KUKA KRL program: EPS_2_25730_SANINSPMH_A_20250909085212.src

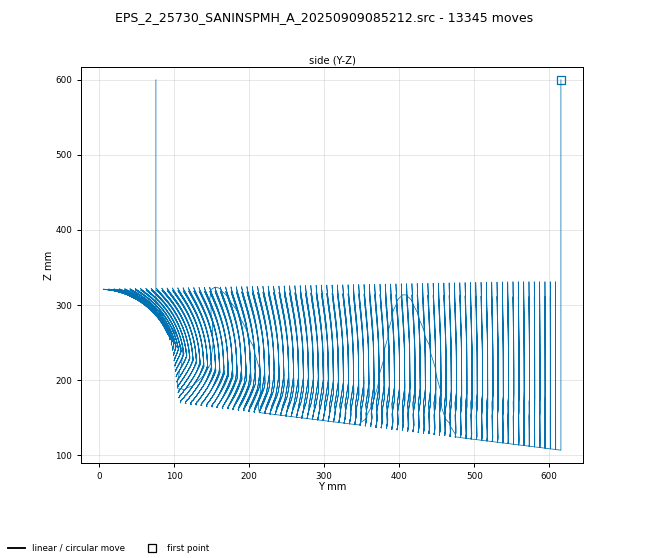
[picture p0: tool path of EPS_2_25730_SANINSPMH_A_20250909085212.src, 13345 of 13347 moves have a stored position in this frame; points joined in program order, loops and branches not executed]
&ACCESS RVP
&REL 4
&COMMENT QRS 19112012
&PARAM EDITMASK = *
DEF PART()
EXT BAS (BAS_COMMAND :IN,REAL :IN )
INT I
BAS (#INITMOV,0 )

;KUKA QRS Post kuka4.cps  Date:22-06-2017 !

File_ID=2820

QRS_PRE_INIT()

;Init var - Until changes are made in qrs_pre_init
Outlet_Square_prg=0
Inlet_1_Square_prg=0
Inlet_2_Square_prg=0
Inlet_3_Square_prg=0
Inlet_4_Square_prg=0
Inlet_5_Square_prg=0

Outlet_1={X 0.000, Y 552.020, Z 256.000, B 0.000, E1 0.000 }
Inlet_1={X 0.000, Y 553.440, Z 236.000, B 0.000, E1 180.000 }
Outlet_1_type=150
Inlet_1_type=150
;QRS#1=Sidecore dimensions
;QRS#2=150-6" PVC SDR 28
;QRS#3=150-6" PVC SDR 28
;QRS#4=
;QRS#5=
;QRS#6=
;QRS#7=
;QRS#8=
;QRS#9=10-06 PSX
;QRS#10=10-06 PSX
;QRS#11=
;QRS#12=
;QRS#13=
;QRS#14=
;QRS#15=
;QRS#16=1220x127x610 2'
;QRS#17=EPS Height
;QRS#18=331
;QRS#19=*
;QRS#20= UPDATED VERSION 22-06-2017
;QRS#21=*
Outlet_Square=070
Inlet_1_Square=070
Inlet_2_Square=0
Inlet_3_Square=0
Inlet_4_Square=0
Inlet_5_Square=0
Mill_Square=1
Outlet_Square_Prg=203
Inlet_1_Square_prg=203

QRS_INIT()

$ADVANCE=5

; T1
PTP {E1 173.612,E2 173.612}
PTP {X 0,Y 615.5,A -85,B 0,C 180,E1 173.612,E2 173.612,E3 0,E4 0,E5 0,E6 0}
QRS_SPEED_INIT()
LIN {X 0,Y 615.5,Z 600,A -85,B 0,C 180,E1 173.612,E2 173.612,E3 0,E4 0,E5 0,E6 0} C_VEL
LIN {X 0,Y 615.5,Z 116.679,A -85,B 0,C 180,E1 173.612,E2 173.612} C_VEL
LIN {X 0,Y 615.5,Z 108.498,A -85,B 0,C 180,E1 173.612,E2 173.612} C_VEL
LIN {X 0,Y 615.484,Z 106.498,A -85,B 0,C 180,E1 173.425,E2 173.425} C_VEL
LIN {X 0,Y 615.477,Z 106.503,A -85,B 0,C 180,E1 170.801,E2 170.801} C_VEL
LIN {X 0,Y 615.484,Z 106.508,A -85,B 0,C 180,E1 168.139,E2 168.139} C_VEL
LIN {X 0,Y 615.491,Z 106.495,A -85,B 0,C 180,E1 165.451,E2 165.451} C_VEL
LIN {X 0,Y 615.489,Z 106.51,A -85,B 0,C 180,E1 162.729,E2 162.729} C_VEL
LIN {X 0,Y 615.481,Z 106.499,A -85,B 0,C 180,E1 159.967,E2 159.967} C_VEL
LIN {X 0,Y 615.481,Z 106.505,A -85,B 0,C 180,E1 157.155,E2 157.155} C_VEL
LIN {X 0,Y 615.477,Z 106.504,A -85,B 0,C 180,E1 154.433,E2 154.433} C_VEL
LIN {X 0,Y 615.485,Z 106.497,A -85,B 0,C 180,E1 152.085,E2 152.085} C_VEL
LIN {X 0,Y 615.489,Z 106.496,A -85,B 0,C 180,E1 149.84,E2 149.84} C_VEL
LIN {X 0,Y 615.481,Z 106.505,A -85,B 0,C 180,E1 147.542,E2 147.542} C_VEL
LIN {X 0,Y 615.495,Z 106.512,A -85,B 0,C 180,E1 145.185,E2 145.185} C_VEL
LIN {X 0,Y 615.472,Z 106.503,A -85,B 0,C 180,E1 142.757,E2 142.757} C_VEL
LIN {X 0,Y 615.483,Z 106.502,A -85,B 0,C 180,E1 139.912,E2 139.912} C_VEL
LIN {X 0,Y 615.491,Z 106.51,A -85,B 0,C 180,E1 137.647,E2 137.647} C_VEL
LIN {X 0,Y 615.474,Z 106.501,A -85,B 0,C 180,E1 134.93,E2 134.93} C_VEL
LIN {X 0,Y 615.482,Z 106.506,A -85,B 0,C 180,E1 132.079,E2 132.079} C_VEL
LIN {X 0,Y 615.491,Z 106.512,A -85,B 0,C 180,E1 129.75,E2 129.75} C_VEL
LIN {X 0,Y 615.48,Z 106.497,A -85,B 0,C 180,E1 126.936,E2 126.936} C_VEL
LIN {X 0,Y 615.492,Z 106.514,A -85,B 0,C 180,E1 124.022,E2 124.022} C_VEL
LIN {X 0,Y 615.472,Z 106.506,A -85,B 0,C 180,E1 121.686,E2 121.686} C_VEL
LIN {X 0,Y 615.473,Z 106.5,A -85,B 0,C 180,E1 119.407,E2 119.407} C_VEL
LIN {X 0,Y 615.493,Z 106.51,A -85,B 0,C 180,E1 116.444,E2 116.444} C_VEL
LIN {X 0,Y 615.472,Z 106.506,A -85,B 0,C 180,E1 114.005,E2 114.005} C_VEL
LIN {X 0,Y 615.485,Z 106.496,A -85,B 0,C 180,E1 111.432,E2 111.432} C_VEL
LIN {X 0,Y 615.499,Z 106.666,A -85,B 0,C 180,E1 108.545,E2 108.545} C_VEL
LIN {X 0,Y 615.476,Z 120.496,A -85,B 0,C 180,E1 105.906,E2 105.906} C_VEL
LIN {X 0,Y 615.489,Z 134.92,A -85,B 0,C 180,E1 103.201,E2 103.201} C_VEL
LIN {X 0,Y 615.474,Z 149.332,A -85,B 0,C 180,E1 100.527,E2 100.527} C_VEL
LIN {X 0,Y 615.496,Z 152.049,A -85,B 0,C 180,E1 100.091,E2 100.091} C_VEL
LIN {X 0,Y 615.495,Z 154.32,A -85,B 0,C 180,E1 100.028,E2 100.028} C_VEL
LIN {X 0,Y 615.496,Z 227.7,A -85,B 0,C 180,E1 99.157,E2 99.157} C_VEL
LIN {X 0,Y 615.497,Z 235.887,A -85,B 0,C 180,E1 98.992,E2 98.992} C_VEL
LIN {X 0,Y 615.497,Z 244.447,A -85,B 0,C 180,E1 98.743,E2 98.743} C_VEL
LIN {X 0,Y 615.497,Z 252.059,A -85,B 0,C 180,E1 98.454,E2 98.454} C_VEL
LIN {X 0,Y 615.499,Z 260.579,A -85,B 0,C 180,E1 98.041,E2 98.041} C_VEL
LIN {X 0,Y 615.489,Z 268.747,A -85,B 0,C 180,E1 97.546,E2 97.546} C_VEL
LIN {X 0,Y 615.492,Z 275.387,A -85,B 0,C 180,E1 97.058,E2 97.058} C_VEL
LIN {X 0,Y 615.498,Z 281.183,A -85,B 0,C 180,E1 96.557,E2 96.557} C_VEL
LIN {X 0,Y 615.499,Z 287.533,A -85,B 0,C 180,E1 95.899,E2 95.899} C_VEL
LIN {X 0,Y 615.495,Z 293.983,A -85,B 0,C 180,E1 95.077,E2 95.077} C_VEL
LIN {X 0,Y 615.491,Z 299.122,A -85,B 0,C 180,E1 94.257,E2 94.257} C_VEL
LIN {X 0,Y 615.493,Z 303.886,A -85,B 0,C 180,E1 93.273,E2 93.273} C_VEL
LIN {X 0,Y 615.493,Z 306.2,A -85,B 0,C 180,E1 92.618,E2 92.618} C_VEL
LIN {X 0,Y 615.499,Z 307.976,A -85,B 0,C 180,E1 91.963,E2 91.963} C_VEL
LIN {X 0,Y 615.492,Z 309.266,A -85,B 0,C 180,E1 91.309,E2 91.309} C_VEL
LIN {X 0,Y 615.491,Z 310.083,A -85,B 0,C 180,E1 90.654,E2 90.654} C_VEL
LIN {X 0,Y 615.492,Z 310.384,A -85,B 0,C 180,E1 90,E2 90} C_VEL
LIN {X 0,Y 615.492,Z 310.125,A -85,B 0,C 180,E1 89.346,E2 89.346} C_VEL
LIN {X 0,Y 615.494,Z 309.394,A -85,B 0,C 180,E1 88.692,E2 88.692} C_VEL
LIN {X 0,Y 615.499,Z 308.195,A -85,B 0,C 180,E1 88.037,E2 88.037} C_VEL
LIN {X 0,Y 615.49,Z 305.377,A -85,B 0,C 180,E1 87.055,E2 87.055} C_VEL
LIN {X 0,Y 615.492,Z 302.81,A -85,B 0,C 180,E1 86.4,E2 86.4} C_VEL
LIN {X 0,Y 615.495,Z 297.744,A -85,B 0,C 180,E1 85.416,E2 85.416} C_VEL
LIN {X 0,Y 615.496,Z 292.289,A -85,B 0,C 180,E1 84.595,E2 84.595} C_VEL
LIN {X 0,Y 615.497,Z 285.454,A -85,B 0,C 180,E1 83.773,E2 83.773} C_VEL
LIN {X 0,Y 615.497,Z 278.42,A -85,B 0,C 180,E1 83.1,E2 83.1} C_VEL
LIN {X 0,Y 615.491,Z 270.073,A -85,B 0,C 180,E1 82.455,E2 82.455} C_VEL
LIN {X 0,Y 615.499,Z 262.197,A -85,B 0,C 180,E1 81.96,E2 81.96} C_VEL
LIN {X 0,Y 615.497,Z 254.076,A -85,B 0,C 180,E1 81.546,E2 81.546} C_VEL
LIN {X 0,Y 615.497,Z 245.865,A -85,B 0,C 180,E1 81.216,E2 81.216} C_VEL
LIN {X 0,Y 615.497,Z 237.842,A -85,B 0,C 180,E1 80.967,E2 80.967} C_VEL
LIN {X 0,Y 615.5,Z 228.165,A -85,B 0,C 180,E1 80.76,E2 80.76} C_VEL
LIN {X 0,Y 615.494,Z 152.561,A -85,B 0,C 180,E1 79.847,E2 79.847} C_VEL
LIN {X 0,Y 615.489,Z 151.218,A -85,B 0,C 180,E1 79.723,E2 79.723} C_VEL
LIN {X 0,Y 615.475,Z 137.207,A -85,B 0,C 180,E1 77.134,E2 77.134} C_VEL
LIN {X 0,Y 615.486,Z 122.781,A -85,B 0,C 180,E1 74.435,E2 74.435} C_VEL
LIN {X 0,Y 615.497,Z 108.44,A -85,B 0,C 180,E1 71.719,E2 71.719} C_VEL
LIN {X 0,Y 615.493,Z 106.562,A -85,B 0,C 180,E1 71.311,E2 71.311} C_VEL
LIN {X 0,Y 615.484,Z 106.497,A -85,B 0,C 180,E1 68.568,E2 68.568} C_VEL
LIN {X 0,Y 615.48,Z 106.51,A -85,B 0,C 180,E1 65.728,E2 65.728} C_VEL
LIN {X 0,Y 615.486,Z 106.497,A -85,B 0,C 180,E1 62.823,E2 62.823} C_VEL
LIN {X 0,Y 615.467,Z 106.506,A -85,B 0,C 180,E1 60.209,E2 60.209} C_VEL
LIN {X 0,Y 615.488,Z 106.506,A -85,B 0,C 180,E1 57.543,E2 57.543} C_VEL
LIN {X 0,Y 615.496,Z 106.495,A -85,B 0,C 180,E1 55.186,E2 55.186} C_VEL
LIN {X 0,Y 615.468,Z 106.501,A -85,B 0,C 180,E1 52.757,E2 52.757} C_VEL
LIN {X 0,Y 615.49,Z 106.508,A -85,B 0,C 180,E1 49.911,E2 49.911} C_VEL
LIN {X 0,Y 615.469,Z 106.502,A -85,B 0,C 180,E1 46.955,E2 46.955} C_VEL
LIN {X 0,Y 615.49,Z 106.508,A -85,B 0,C 180,E1 44.149,E2 44.149} C_VEL
LIN {X 0,Y 615.485,Z 106.496,A -85,B 0,C 180,E1 41.474,E2 41.474} C_VEL
LIN {X 0,Y 615.475,Z 106.507,A -85,B 0,C 180,E1 38.905,E2 38.905} C_VEL
LIN {X 0,Y 615.484,Z 106.509,A -85,B 0,C 180,E1 36.425,E2 36.425} C_VEL
LIN {X 0,Y 615.487,Z 106.498,A -85,B 0,C 180,E1 34.022,E2 34.022} C_VEL
LIN {X 0,Y 615.481,Z 106.498,A -85,B 0,C 180,E1 31.686,E2 31.686} C_VEL
LIN {X 0,Y 615.473,Z 106.504,A -85,B 0,C 180,E1 29.407,E2 29.407} C_VEL
LIN {X 0,Y 615.493,Z 106.512,A -85,B 0,C 180,E1 27.047,E2 27.047} C_VEL
LIN {X 0,Y 615.485,Z 106.496,A -85,B 0,C 180,E1 24.008,E2 24.008} C_VEL
LIN {X 0,Y 615.483,Z 106.509,A -85,B 0,C 180,E1 21.432,E2 21.432} C_VEL
LIN {X 0,Y 615.486,Z 106.498,A -85,B 0,C 180,E1 18.605,E2 18.605} C_VEL
LIN {X 0,Y 615.474,Z 106.504,A -85,B 0,C 180,E1 15.906,E2 15.906} C_VEL
LIN {X 0,Y 615.479,Z 106.507,A -85,B 0,C 180,E1 13.201,E2 13.201} C_VEL
LIN {X 0,Y 615.486,Z 106.496,A -85,B 0,C 180,E1 10.527,E2 10.527} C_VEL
LIN {X 0,Y 615.486,Z 106.51,A -85,B 0,C 180,E1 7.876,E2 7.876} C_VEL
LIN {X 0,Y 615.479,Z 106.501,A -85,B 0,C 180,E1 5.241,E2 5.241} C_VEL
LIN {X 0,Y 615.482,Z 106.499,A -85,B 0,C 180,E1 2.618,E2 2.618} C_VEL
LIN {X 0,Y 615.487,Z 106.515,A -85,B 0,C 180,E1 0,E2 0} C_VEL
LIN {X 0,Y 615.481,Z 106.499,A -85,B 0,C 180,E1 -2.618,E2 -2.618} C_VEL
LIN {X 0,Y 615.481,Z 106.502,A -85,B 0,C 180,E1 -5.241,E2 -5.241} C_VEL
LIN {X 0,Y 615.485,Z 106.509,A -85,B 0,C 180,E1 -7.876,E2 -7.876} C_VEL
LIN {X 0,Y 615.485,Z 106.496,A -85,B 0,C 180,E1 -10.527,E2 -10.527} C_VEL
LIN {X 0,Y 615.485,Z 106.507,A -85,B 0,C 180,E1 -13.201,E2 -13.201} C_VEL
LIN {X 0,Y 615.474,Z 106.503,A -85,B 0,C 180,E1 -15.905,E2 -15.905} C_VEL
LIN {X 0,Y 615.486,Z 106.499,A -85,B 0,C 180,E1 -18.646,E2 -18.646} C_VEL
LIN {X 0,Y 615.479,Z 106.508,A -85,B 0,C 180,E1 -21.432,E2 -21.432} C_VEL
LIN {X 0,Y 615.489,Z 106.496,A -85,B 0,C 180,E1 -24.272,E2 -24.272} C_VEL
LIN {X 0,Y 615.477,Z 106.51,A -85,B 0,C 180,E1 -27.178,E2 -27.178} C_VEL
LIN {X 0,Y 615.482,Z 106.497,A -85,B 0,C 180,E1 -29.794,E2 -29.794} C_VEL
LIN {X 0,Y 615.486,Z 106.506,A -85,B 0,C 180,E1 -32.457,E2 -32.457} C_VEL
LIN {X 0,Y 615.485,Z 106.51,A -85,B 0,C 180,E1 -34.815,E2 -34.815} C_VEL
LIN {X 0,Y 615.469,Z 106.502,A -85,B 0,C 180,E1 -37.243,E2 -37.243} C_VEL
LIN {X 0,Y 615.486,Z 106.504,A -85,B 0,C 180,E1 -40.089,E2 -40.089} C_VEL
LIN {X 0,Y 615.499,Z 106.513,A -85,B 0,C 180,E1 -42.352,E2 -42.352} C_VEL
LIN {X 0,Y 615.47,Z 106.5,A -85,B 0,C 180,E1 -45.07,E2 -45.07} C_VEL
LIN {X 0,Y 615.49,Z 106.507,A -85,B 0,C 180,E1 -47.919,E2 -47.919} C_VEL
LIN {X 0,Y 615.48,Z 106.51,A -85,B 0,C 180,E1 -50.25,E2 -50.25} C_VEL
LIN {X 0,Y 615.478,Z 106.498,A -85,B 0,C 180,E1 -53.064,E2 -53.064} C_VEL
LIN {X 0,Y 615.485,Z 106.511,A -85,B 0,C 180,E1 -55.978,E2 -55.978} C_VEL
LIN {X 0,Y 615.461,Z 106.506,A -85,B 0,C 180,E1 -58.313,E2 -58.313} C_VEL
LIN {X 0,Y 615.469,Z 106.5,A -85,B 0,C 180,E1 -60.593,E2 -60.593} C_VEL
LIN {X 0,Y 615.497,Z 106.497,A -85,B 0,C 180,E1 -62.953,E2 -62.953} C_VEL
LIN {X 0,Y 615.475,Z 106.509,A -85,B 0,C 180,E1 -65.728,E2 -65.728} C_VEL
LIN {X 0,Y 615.463,Z 106.507,A -85,B 0,C 180,E1 -67.863,E2 -67.863} C_VEL
LIN {X 0,Y 615.494,Z 106.696,A -85,B 0,C 180,E1 -69.398,E2 -69.398} C_VEL
LIN {X 0,Y 615.489,Z 122.513,A -85,B 0,C 180,E1 -72.043,E2 -72.043} C_VEL
LIN {X 0,Y 615.468,Z 140.241,A -85,B 0,C 180,E1 -74.943,E2 -74.943} C_VEL
LIN {X 0,Y 615.465,Z 155.869,A -85,B 0,C 180,E1 -77.47,E2 -77.47} C_VEL
LIN {X 0,Y 615.491,Z 170.941,A -85,B 0,C 180,E1 -79.847,E2 -79.847} C_VEL
LIN {X 0,Y 615.489,Z 172.866,A -85,B 0,C 180,E1 -79.91,E2 -79.91} C_VEL
LIN {X 0,Y 615.493,Z 247.945,A -85,B 0,C 180,E1 -80.801,E2 -80.801} C_VEL
LIN {X 0,Y 615.496,Z 257.699,A -85,B 0,C 180,E1 -81.009,E2 -81.009} C_VEL
LIN {X 0,Y 615.499,Z 268.156,A -85,B 0,C 180,E1 -81.34,E2 -81.34} C_VEL
LIN {X 0,Y 615.497,Z 278.43,A -85,B 0,C 180,E1 -81.794,E2 -81.794} C_VEL
LIN {X 0,Y 615.493,Z 288.2,A -85,B 0,C 180,E1 -82.372,E2 -82.372} C_VEL
LIN {X 0,Y 615.494,Z 295.936,A -85,B 0,C 180,E1 -82.942,E2 -82.942} C_VEL
LIN {X 0,Y 615.497,Z 303.336,A -85,B 0,C 180,E1 -83.608,E2 -83.608} C_VEL
LIN {X 0,Y 615.498,Z 310.739,A -85,B 0,C 180,E1 -84.43,E2 -84.43} C_VEL
LIN {X 0,Y 615.497,Z 316.534,A -85,B 0,C 180,E1 -85.252,E2 -85.252} C_VEL
LIN {X 0,Y 615.496,Z 321.101,A -85,B 0,C 180,E1 -86.072,E2 -86.072} C_VEL
LIN {X 0,Y 615.492,Z 324.069,A -85,B 0,C 180,E1 -86.727,E2 -86.727} C_VEL
LIN {X 0,Y 615.494,Z 326.357,A -85,B 0,C 180,E1 -87.382,E2 -87.382} C_VEL
LIN {X 0,Y 615.499,Z 328.085,A -85,B 0,C 180,E1 -88.037,E2 -88.037} C_VEL
LIN {X 0,Y 615.493,Z 329.33,A -85,B 0,C 180,E1 -88.692,E2 -88.692} C_VEL
LIN {X 0,Y 615.491,Z 330.104,A -85,B 0,C 180,E1 -89.346,E2 -89.346} C_VEL
LIN {X 0,Y 615.491,Z 330.389,A -85,B 0,C 180,E1 -90,E2 -90} C_VEL
LIN {X 0,Y 615.492,Z 330.104,A -85,B 0,C 180,E1 -90.654,E2 -90.654} C_VEL
LIN {X 0,Y 615.493,Z 329.33,A -85,B 0,C 180,E1 -91.309,E2 -91.309} C_VEL
LIN {X 0,Y 615.499,Z 328.085,A -85,B 0,C 180,E1 -91.963,E2 -91.963} C_VEL
LIN {X 0,Y 615.488,Z 325.22,A -85,B 0,C 180,E1 -92.946,E2 -92.946} C_VEL
LIN {X 0,Y 615.491,Z 322.603,A -85,B 0,C 180,E1 -93.601,E2 -93.601} C_VEL
LIN {X 0,Y 615.495,Z 317.481,A -85,B 0,C 180,E1 -94.585,E2 -94.585} C_VEL
LIN {X 0,Y 615.495,Z 311.967,A -85,B 0,C 180,E1 -95.406,E2 -95.406} C_VEL
LIN {X 0,Y 615.498,Z 305.016,A -85,B 0,C 180,E1 -96.228,E2 -96.228} C_VEL
LIN {X 0,Y 615.496,Z 297.858,A -85,B 0,C 180,E1 -96.901,E2 -96.901} C_VEL
LIN {X 0,Y 615.488,Z 290.619,A -85,B 0,C 180,E1 -97.463,E2 -97.463} C_VEL
LIN {X 0,Y 615.498,Z 282.865,A -85,B 0,C 180,E1 -97.958,E2 -97.958} C_VEL
LIN {X 0,Y 615.498,Z 274.91,A -85,B 0,C 180,E1 -98.371,E2 -98.371} C_VEL
LIN {X 0,Y 615.497,Z 265.75,A -85,B 0,C 180,E1 -98.743,E2 -98.743} C_VEL
LIN {X 0,Y 615.496,Z 257.686,A -85,B 0,C 180,E1 -98.992,E2 -98.992} C_VEL
LIN {X 0,Y 615.493,Z 247.925,A -85,B 0,C 180,E1 -99.199,E2 -99.199} C_VEL
LIN {X 0,Y 615.49,Z 171.745,A -85,B 0,C 180,E1 -100.111,E2 -100.111} C_VEL
LIN {X 0,Y 615.489,Z 170.51,A -85,B 0,C 180,E1 -100.194,E2 -100.194} C_VEL
LIN {X 0,Y 615.49,Z 153.783,A -85,B 0,C 180,E1 -102.866,E2 -102.866} C_VEL
LIN {X 0,Y 615.481,Z 136.068,A -85,B 0,C 180,E1 -105.735,E2 -105.735} C_VEL
LIN {X 0,Y 615.487,Z 120.566,A -85,B 0,C 180,E1 -108.278,E2 -108.278} C_VEL
LIN {X 0,Y 615.494,Z 106.695,A -85,B 0,C 180,E1 -110.602,E2 -110.602} C_VEL
LIN {X 0,Y 615.491,Z 106.506,A -85,B 0,C 180,E1 -112.844,E2 -112.844} C_VEL
LIN {X 0,Y 615.461,Z 106.503,A -85,B 0,C 180,E1 -115.717,E2 -115.717} C_VEL
LIN {X 0,Y 615.497,Z 106.511,A -85,B 0,C 180,E1 -118.452,E2 -118.452} C_VEL
LIN {X 0,Y 615.48,Z 106.498,A -85,B 0,C 180,E1 -121.085,E2 -121.085} C_VEL
LIN {X 0,Y 615.463,Z 106.504,A -85,B 0,C 180,E1 -123.531,E2 -123.531} C_VEL
LIN {X 0,Y 615.475,Z 106.509,A -85,B 0,C 180,E1 -125.832,E2 -125.832} C_VEL
LIN {X 0,Y 615.488,Z 106.514,A -85,B 0,C 180,E1 -128.069,E2 -128.069} C_VEL
LIN {X 0,Y 615.487,Z 106.498,A -85,B 0,C 180,E1 -130.607,E2 -130.607} C_VEL
LIN {X 0,Y 615.465,Z 106.504,A -85,B 0,C 180,E1 -133.247,E2 -133.247} C_VEL
LIN {X 0,Y 615.489,Z 106.506,A -85,B 0,C 180,E1 -136.003,E2 -136.003} C_VEL
LIN {X 0,Y 615.484,Z 106.497,A -85,B 0,C 180,E1 -138.526,E2 -138.526} C_VEL
LIN {X 0,Y 615.47,Z 106.506,A -85,B 0,C 180,E1 -141.094,E2 -141.094} C_VEL
LIN {X 0,Y 615.486,Z 106.511,A -85,B 0,C 180,E1 -143.575,E2 -143.575} C_VEL
LIN {X 0,Y 615.474,Z 106.499,A -85,B 0,C 180,E1 -146.468,E2 -146.468} C_VEL
LIN {X 0,Y 615.486,Z 106.51,A -85,B 0,C 180,E1 -149.08,E2 -149.08} C_VEL
LIN {X 0,Y 615.483,Z 106.497,A -85,B 0,C 180,E1 -152.085,E2 -152.085} C_VEL
LIN {X 0,Y 615.492,Z 106.514,A -85,B 0,C 180,E1 -155.009,E2 -155.009} C_VEL
LIN {X 0,Y 615.485,Z 106.496,A -85,B 0,C 180,E1 -157.864,E2 -157.864} C_VEL
LIN {X 0,Y 615.488,Z 106.51,A -85,B 0,C 180,E1 -160.662,E2 -160.662} C_VEL
LIN {X 0,Y 615.488,Z 106.496,A -85,B 0,C 180,E1 -163.569,E2 -163.569} C_VEL
LIN {X 0,Y 615.473,Z 106.505,A -85,B 0,C 180,E1 -166.126,E2 -166.126} C_VEL
LIN {X 0,Y 615.485,Z 106.506,A -85,B 0,C 180,E1 -168.807,E2 -168.807} C_VEL
LIN {X 0,Y 615.486,Z 106.496,A -85,B 0,C 180,E1 -171.463,E2 -171.463} C_VEL
LIN {X 0,Y 615.485,Z 106.509,A -85,B 0,C 180,E1 -174.102,E2 -174.102} C_VEL
LIN {X 0,Y 615.479,Z 106.502,A -85,B 0,C 180,E1 -176.727,E2 -176.727} C_VEL
LIN {X 0,Y 615.479,Z 106.499,A -85,B 0,C 180,E1 -179.346,E2 -179.346} C_VEL
LIN {X 0,Y 615.496,Z 106.512,A -85,B 0,C 180,E1 -181.963,E2 -181.963} C_VEL
LIN {X 0,Y 615.484,Z 106.498,A -85,B 0,C 180,E1 -184.585,E2 -184.585} C_VEL
LIN {X 0,Y 615.484,Z 106.498,A -85,B 0,C 180,E1 -186.575,E2 -186.575} C_VEL
LIN {X 0,Y 614.803,Z 106.649,A -85,B 0,C 180,E1 -187.121,E2 -187.121} C_VEL
LIN {X 0,Y 611.964,Z 107.069,A -85,B 0,C 180,E1 -188.007,E2 -188.007} C_VEL
LIN {X 0,Y 609.574,Z 107.378,A -85,B 0,C 180,E1 -188.719,E2 -188.719} C_VEL
LIN {X 0,Y 608.543,Z 107.494,A -85,B 0,C 180,E1 -189.269,E2 -189.269} C_VEL
LIN {X 0,Y 608.455,Z 107.503,A -85,B 0,C 180,E1 -189.455,E2 -189.455} C_VEL
LIN {X 0,Y 608.462,Z 107.503,A -85,B 0,C 180,E1 -192,E2 -192} C_VEL
LIN {X 0,Y 608.478,Z 107.498,A -85,B 0,C 180,E1 -194.721,E2 -194.721} C_VEL
LIN {X 0,Y 608.453,Z 107.51,A -85,B 0,C 180,E1 -197.477,E2 -197.477} C_VEL
LIN {X 0,Y 608.46,Z 107.499,A -85,B 0,C 180,E1 -200.274,E2 -200.274} C_VEL
LIN {X 0,Y 608.46,Z 107.5,A -85,B 0,C 180,E1 -202.476,E2 -202.476} C_VEL
LIN {X 0,Y 608.456,Z 107.502,A -85,B 0,C 180,E1 -204.571,E2 -204.571} C_VEL
LIN {X 0,Y 608.484,Z 107.504,A -85,B 0,C 180,E1 -207.208,E2 -207.208} C_VEL
LIN {X 0,Y 608.467,Z 107.498,A -85,B 0,C 180,E1 -209.971,E2 -209.971} C_VEL
LIN {X 0,Y 608.452,Z 107.51,A -85,B 0,C 180,E1 -212.88,E2 -212.88} C_VEL
LIN {X 0,Y 608.444,Z 107.504,A -85,B 0,C 180,E1 -215.278,E2 -215.278} C_VEL
LIN {X 0,Y 608.464,Z 107.503,A -85,B 0,C 180,E1 -218.24,E2 -218.24} C_VEL
LIN {X 0,Y 608.456,Z 107.5,A -85,B 0,C 180,E1 -221.342,E2 -221.342} C_VEL
LIN {X 0,Y 608.452,Z 107.508,A -85,B 0,C 180,E1 -224.263,E2 -224.263} C_VEL
LIN {X 0,Y 608.441,Z 107.502,A -85,B 0,C 180,E1 -227.039,E2 -227.039} C_VEL
LIN {X 0,Y 608.454,Z 107.503,A -85,B 0,C 180,E1 -229.697,E2 -229.697} C_VEL
LIN {X 0,Y 608.465,Z 107.506,A -85,B 0,C 180,E1 -232.253,E2 -232.253} C_VEL
LIN {X 0,Y 608.485,Z 107.496,A -85,B 0,C 180,E1 -235.09,E2 -235.09} C_VEL
LIN {X 0,Y 608.464,Z 107.509,A -85,B 0,C 180,E1 -237.905,E2 -237.905} C_VEL
LIN {X 0,Y 608.458,Z 107.503,A -85,B 0,C 180,E1 -240.22,E2 -240.22} C_VEL
LIN {X 0,Y 608.482,Z 107.497,A -85,B 0,C 180,E1 -242.792,E2 -242.792} C_VEL
LIN {X 0,Y 608.472,Z 107.504,A -85,B 0,C 180,E1 -245.849,E2 -245.849} C_VEL
LIN {X 0,Y 608.464,Z 107.499,A -85,B 0,C 180,E1 -248.308,E2 -248.308} C_VEL
LIN {X 0,Y 608.49,Z 107.574,A -85,B 0,C 180,E1 -251.379,E2 -251.379} C_VEL
LIN {X 0,Y 608.48,Z 120.639,A -85,B 0,C 180,E1 -253.907,E2 -253.907} C_VEL
LIN {X 0,Y 608.477,Z 135.127,A -85,B 0,C 180,E1 -256.644,E2 -256.644} C_VEL
LIN {X 0,Y 608.424,Z 149.617,A -85,B 0,C 180,E1 -259.349,E2 -259.349} C_VEL
LIN {X 0,Y 608.471,Z 152.233,A -85,B 0,C 180,E1 -259.792,E2 -259.792} C_VEL
LIN {X 0,Y 608.525,Z 154.822,A -85,B 0,C 180,E1 -259.856,E2 -259.856} C_VEL
LIN {X 0,Y 608.511,Z 228.245,A -85,B 0,C 180,E1 -260.737,E2 -260.737} C_VEL
LIN {X 0,Y 608.512,Z 237.948,A -85,B 0,C 180,E1 -260.946,E2 -260.946} C_VEL
LIN {X 0,Y 608.499,Z 249.535,A -85,B 0,C 180,E1 -261.323,E2 -261.323} C_VEL
LIN {X 0,Y 608.479,Z 259.431,A -85,B 0,C 180,E1 -261.782,E2 -261.782} C_VEL
LIN {X 0,Y 608.473,Z 267.884,A -85,B 0,C 180,E1 -262.283,E2 -262.283} C_VEL
LIN {X 0,Y 608.46,Z 275.853,A -85,B 0,C 180,E1 -262.867,E2 -262.867} C_VEL
LIN {X 0,Y 608.467,Z 282.902,A -85,B 0,C 180,E1 -263.496,E2 -263.496} C_VEL
LIN {X 0,Y 608.458,Z 289.394,A -85,B 0,C 180,E1 -264.199,E2 -264.199} C_VEL
LIN {X 0,Y 608.437,Z 295.641,A -85,B 0,C 180,E1 -265.03,E2 -265.03} C_VEL
LIN {X 0,Y 608.434,Z 301.424,A -85,B 0,C 180,E1 -266.026,E2 -266.026} C_VEL
LIN {X 0,Y 608.447,Z 305.63,A -85,B 0,C 180,E1 -267.02,E2 -267.02} C_VEL
LIN {X 0,Y 608.443,Z 308.569,A -85,B 0,C 180,E1 -268.014,E2 -268.014} C_VEL
LIN {X 0,Y 608.445,Z 309.87,A -85,B 0,C 180,E1 -268.676,E2 -268.676} C_VEL
LIN {X 0,Y 608.434,Z 310.692,A -85,B 0,C 180,E1 -269.338,E2 -269.338} C_VEL
LIN {X 0,Y 608.432,Z 310.995,A -85,B 0,C 180,E1 -270,E2 -270} C_VEL
LIN {X 0,Y 608.435,Z 310.735,A -85,B 0,C 180,E1 -270.662,E2 -270.662} C_VEL
LIN {X 0,Y 608.446,Z 309.998,A -85,B 0,C 180,E1 -271.324,E2 -271.324} C_VEL
LIN {X 0,Y 608.443,Z 308.787,A -85,B 0,C 180,E1 -271.986,E2 -271.986} C_VEL
LIN {X 0,Y 608.445,Z 305.942,A -85,B 0,C 180,E1 -272.979,E2 -272.979} C_VEL
LIN {X 0,Y 608.446,Z 303.353,A -85,B 0,C 180,E1 -273.642,E2 -273.642} C_VEL
LIN {X 0,Y 608.445,Z 298.245,A -85,B 0,C 180,E1 -274.638,E2 -274.638} C_VEL
LIN {X 0,Y 608.461,Z 292.75,A -85,B 0,C 180,E1 -275.468,E2 -275.468} C_VEL
LIN {X 0,Y 608.454,Z 285.15,A -85,B 0,C 180,E1 -276.374,E2 -276.374} C_VEL
LIN {X 0,Y 608.463,Z 276.951,A -85,B 0,C 180,E1 -277.132,E2 -277.132} C_VEL
LIN {X 0,Y 608.473,Z 269.202,A -85,B 0,C 180,E1 -277.716,E2 -277.716} C_VEL
LIN {X 0,Y 608.48,Z 261.037,A -85,B 0,C 180,E1 -278.217,E2 -278.217} C_VEL
LIN {X 0,Y 608.484,Z 250.677,A -85,B 0,C 180,E1 -278.719,E2 -278.719} C_VEL
LIN {X 0,Y 608.511,Z 239.038,A -85,B 0,C 180,E1 -279.116,E2 -279.116} C_VEL
LIN {X 0,Y 608.524,Z 228.648,A -85,B 0,C 180,E1 -279.347,E2 -279.347} C_VEL
LIN {X 0,Y 608.514,Z 189.347,A -85,B 0,C 180,E1 -279.829,E2 -279.829} C_VEL
LIN {X 0,Y 608.489,Z 152.717,A -85,B 0,C 180,E1 -280.271,E2 -280.271} C_VEL
LIN {X 0,Y 608.456,Z 151.482,A -85,B 0,C 180,E1 -280.397,E2 -280.397} C_VEL
LIN {X 0,Y 608.447,Z 137.42,A -85,B 0,C 180,E1 -283.017,E2 -283.017} C_VEL
LIN {X 0,Y 608.456,Z 122.926,A -85,B 0,C 180,E1 -285.75,E2 -285.75} C_VEL
LIN {X 0,Y 608.491,Z 107.915,A -85,B 0,C 180,E1 -288.622,E2 -288.622} C_VEL
LIN {X 0,Y 608.462,Z 107.507,A -85,B 0,C 180,E1 -288.869,E2 -288.869} C_VEL
LIN {X 0,Y 608.461,Z 107.499,A -85,B 0,C 180,E1 -291.692,E2 -291.692} C_VEL
LIN {X 0,Y 608.453,Z 107.509,A -85,B 0,C 180,E1 -294.571,E2 -294.571} C_VEL
LIN {X 0,Y 608.443,Z 107.502,A -85,B 0,C 180,E1 -297.518,E2 -297.518} C_VEL
LIN {X 0,Y 608.457,Z 107.505,A -85,B 0,C 180,E1 -299.97,E2 -299.97} C_VEL
LIN {X 0,Y 608.452,Z 107.501,A -85,B 0,C 180,E1 -302.88,E2 -302.88} C_VEL
LIN {X 0,Y 608.437,Z 107.503,A -85,B 0,C 180,E1 -305.278,E2 -305.278} C_VEL
LIN {X 0,Y 608.467,Z 107.504,A -85,B 0,C 180,E1 -308.24,E2 -308.24} C_VEL
LIN {X 0,Y 608.449,Z 107.503,A -85,B 0,C 180,E1 -311.341,E2 -311.341} C_VEL
LIN {X 0,Y 608.453,Z 107.503,A -85,B 0,C 180,E1 -314.263,E2 -314.263} C_VEL
LIN {X 0,Y 608.44,Z 107.504,A -85,B 0,C 180,E1 -317.039,E2 -317.039} C_VEL
LIN {X 0,Y 608.451,Z 107.508,A -85,B 0,C 180,E1 -319.696,E2 -319.696} C_VEL
LIN {X 0,Y 608.465,Z 107.499,A -85,B 0,C 180,E1 -322.253,E2 -322.253} C_VEL
LIN {X 0,Y 608.443,Z 107.503,A -85,B 0,C 180,E1 -324.722,E2 -324.722} C_VEL
LIN {X 0,Y 608.459,Z 107.505,A -85,B 0,C 180,E1 -327.478,E2 -327.478} C_VEL
LIN {X 0,Y 608.468,Z 107.498,A -85,B 0,C 180,E1 -330.22,E2 -330.22} C_VEL
LIN {X 0,Y 608.479,Z 107.503,A -85,B 0,C 180,E1 -332.792,E2 -332.792} C_VEL
LIN {X 0,Y 608.479,Z 107.497,A -85,B 0,C 180,E1 -335.847,E2 -335.847} C_VEL
LIN {X 0,Y 608.467,Z 107.501,A -85,B 0,C 180,E1 -338.308,E2 -338.308} C_VEL
LIN {X 0,Y 608.47,Z 107.5,A -85,B 0,C 180,E1 -341.283,E2 -341.283} C_VEL
LIN {X 0,Y 608.454,Z 107.501,A -85,B 0,C 180,E1 -343.906,E2 -343.906} C_VEL
LIN {X 0,Y 608.457,Z 107.507,A -85,B 0,C 180,E1 -346.643,E2 -346.643} C_VEL
LIN {X 0,Y 608.464,Z 107.499,A -85,B 0,C 180,E1 -349.35,E2 -349.35} C_VEL
LIN {X 0,Y 608.477,Z 107.503,A -85,B 0,C 180,E1 -352.033,E2 -352.033} C_VEL
LIN {X 0,Y 608.46,Z 107.502,A -85,B 0,C 180,E1 -354.698,E2 -354.698} C_VEL
LIN {X 0,Y 608.473,Z 107.499,A -85,B 0,C 180,E1 -357.352,E2 -357.352} C_VEL
LIN {X 0,Y 608.477,Z 107.507,A -85,B 0,C 180,E1 -360,E2 -360} C_VEL
LIN {X 0,Y 608.472,Z 107.498,A -85,B 0,C 180,E1 -362.648,E2 -362.648} C_VEL
LIN {X 0,Y 608.461,Z 107.502,A -85,B 0,C 180,E1 -365.302,E2 -365.302} C_VEL
LIN {X 0,Y 608.477,Z 107.503,A -85,B 0,C 180,E1 -367.967,E2 -367.967} C_VEL
LIN {X 0,Y 608.468,Z 107.5,A -85,B 0,C 180,E1 -370.956,E2 -370.956} C_VEL
LIN {X 0,Y 608.46,Z 107.508,A -85,B 0,C 180,E1 -373.356,E2 -373.356} C_VEL
LIN {X 0,Y 608.454,Z 107.501,A -85,B 0,C 180,E1 -376.094,E2 -376.094} C_VEL
LIN {X 0,Y 608.456,Z 107.504,A -85,B 0,C 180,E1 -378.87,E2 -378.87} C_VEL
LIN {X 0,Y 608.464,Z 107.501,A -85,B 0,C 180,E1 -381.692,E2 -381.692} C_VEL
LIN {X 0,Y 608.457,Z 107.503,A -85,B 0,C 180,E1 -384.571,E2 -384.571} C_VEL
LIN {X 0,Y 608.444,Z 107.503,A -85,B 0,C 180,E1 -387.518,E2 -387.518} C_VEL
LIN {X 0,Y 608.466,Z 107.499,A -85,B 0,C 180,E1 -389.972,E2 -389.972} C_VEL
LIN {X 0,Y 608.45,Z 107.508,A -85,B 0,C 180,E1 -392.88,E2 -392.88} C_VEL
LIN {X 0,Y 608.439,Z 107.503,A -85,B 0,C 180,E1 -395.278,E2 -395.278} C_VEL
LIN {X 0,Y 608.466,Z 107.504,A -85,B 0,C 180,E1 -398.241,E2 -398.241} C_VEL
LIN {X 0,Y 608.454,Z 107.5,A -85,B 0,C 180,E1 -401.342,E2 -401.342} C_VEL
LIN {X 0,Y 608.459,Z 107.51,A -85,B 0,C 180,E1 -404.264,E2 -404.264} C_VEL
LIN {X 0,Y 608.437,Z 107.502,A -85,B 0,C 180,E1 -407.039,E2 -407.039} C_VEL
LIN {X 0,Y 608.456,Z 107.504,A -85,B 0,C 180,E1 -409.697,E2 -409.697} C_VEL
LIN {X 0,Y 608.462,Z 107.505,A -85,B 0,C 180,E1 -412.254,E2 -412.254} C_VEL
LIN {X 0,Y 608.484,Z 107.497,A -85,B 0,C 180,E1 -415.09,E2 -415.09} C_VEL
LIN {X 0,Y 608.464,Z 107.507,A -85,B 0,C 180,E1 -417.906,E2 -417.906} C_VEL
LIN {X 0,Y 608.449,Z 107.503,A -85,B 0,C 180,E1 -420.22,E2 -420.22} C_VEL
LIN {X 0,Y 608.481,Z 107.497,A -85,B 0,C 180,E1 -422.792,E2 -422.792} C_VEL
LIN {X 0,Y 608.462,Z 107.502,A -85,B 0,C 180,E1 -425.851,E2 -425.851} C_VEL
LIN {X 0,Y 608.459,Z 107.501,A -85,B 0,C 180,E1 -428.308,E2 -428.308} C_VEL
LIN {X 0,Y 608.506,Z 107.66,A -85,B 0,C 180,E1 -429.312,E2 -429.312} C_VEL
LIN {X 0,Y 608.486,Z 122.58,A -85,B 0,C 180,E1 -431.83,E2 -431.83} C_VEL
LIN {X 0,Y 608.482,Z 139.321,A -85,B 0,C 180,E1 -434.595,E2 -434.595} C_VEL
LIN {X 0,Y 608.446,Z 156.062,A -85,B 0,C 180,E1 -437.323,E2 -437.323} C_VEL
LIN {X 0,Y 608.467,Z 171.122,A -85,B 0,C 180,E1 -439.729,E2 -439.729} C_VEL
LIN {X 0,Y 608.517,Z 173.315,A -85,B 0,C 180,E1 -439.793,E2 -439.793} C_VEL
LIN {X 0,Y 608.504,Z 247.155,A -85,B 0,C 180,E1 -440.674,E2 -440.674} C_VEL
LIN {X 0,Y 608.522,Z 256.421,A -85,B 0,C 180,E1 -440.863,E2 -440.863} C_VEL
LIN {X 0,Y 608.489,Z 264.893,A -85,B 0,C 180,E1 -441.114,E2 -441.114} C_VEL
LIN {X 0,Y 608.502,Z 273.393,A -85,B 0,C 180,E1 -441.448,E2 -441.448} C_VEL
LIN {X 0,Y 608.497,Z 281.723,A -85,B 0,C 180,E1 -441.866,E2 -441.866} C_VEL
LIN {X 0,Y 608.472,Z 289.762,A -85,B 0,C 180,E1 -442.367,E2 -442.367} C_VEL
LIN {X 0,Y 608.453,Z 297.417,A -85,B 0,C 180,E1 -442.951,E2 -442.951} C_VEL
LIN {X 0,Y 608.452,Z 305.439,A -85,B 0,C 180,E1 -443.7,E2 -443.7} C_VEL
LIN {X 0,Y 608.46,Z 312.431,A -85,B 0,C 180,E1 -444.532,E2 -444.532} C_VEL
LIN {X 0,Y 608.431,Z 317.986,A -85,B 0,C 180,E1 -445.362,E2 -445.362} C_VEL
LIN {X 0,Y 608.445,Z 323.147,A -85,B 0,C 180,E1 -446.358,E2 -446.358} C_VEL
LIN {X 0,Y 608.444,Z 325.786,A -85,B 0,C 180,E1 -447.021,E2 -447.021} C_VEL
LIN {X 0,Y 608.443,Z 328.679,A -85,B 0,C 180,E1 -448.014,E2 -448.014} C_VEL
LIN {X 0,Y 608.445,Z 329.934,A -85,B 0,C 180,E1 -448.676,E2 -448.676} C_VEL
LIN {X 0,Y 608.434,Z 330.714,A -85,B 0,C 180,E1 -449.338,E2 -449.338} C_VEL
LIN {X 0,Y 608.431,Z 331,A -85,B 0,C 180,E1 -450,E2 -450} C_VEL
LIN {X 0,Y 608.434,Z 330.714,A -85,B 0,C 180,E1 -450.662,E2 -450.662} C_VEL
LIN {X 0,Y 608.445,Z 329.933,A -85,B 0,C 180,E1 -451.324,E2 -451.324} C_VEL
LIN {X 0,Y 608.443,Z 328.678,A -85,B 0,C 180,E1 -451.986,E2 -451.986} C_VEL
LIN {X 0,Y 608.444,Z 325.785,A -85,B 0,C 180,E1 -452.98,E2 -452.98} C_VEL
LIN {X 0,Y 608.445,Z 323.145,A -85,B 0,C 180,E1 -453.643,E2 -453.643} C_VEL
LIN {X 0,Y 608.431,Z 317.984,A -85,B 0,C 180,E1 -454.638,E2 -454.638} C_VEL
LIN {X 0,Y 608.46,Z 312.429,A -85,B 0,C 180,E1 -455.468,E2 -455.468} C_VEL
LIN {X 0,Y 608.455,Z 304.67,A -85,B 0,C 180,E1 -456.376,E2 -456.376} C_VEL
LIN {X 0,Y 608.453,Z 297.413,A -85,B 0,C 180,E1 -457.05,E2 -457.05} C_VEL
LIN {X 0,Y 608.472,Z 289.758,A -85,B 0,C 180,E1 -457.633,E2 -457.633} C_VEL
LIN {X 0,Y 608.497,Z 281.717,A -85,B 0,C 180,E1 -458.134,E2 -458.134} C_VEL
LIN {X 0,Y 608.502,Z 273.386,A -85,B 0,C 180,E1 -458.552,E2 -458.552} C_VEL
LIN {X 0,Y 608.49,Z 264.884,A -85,B 0,C 180,E1 -458.887,E2 -458.887} C_VEL
LIN {X 0,Y 608.512,Z 255.578,A -85,B 0,C 180,E1 -459.159,E2 -459.159} C_VEL
LIN {X 0,Y 608.51,Z 244.538,A -85,B 0,C 180,E1 -459.368,E2 -459.368} C_VEL
LIN {X 0,Y 608.508,Z 171.945,A -85,B 0,C 180,E1 -460.229,E2 -460.229} C_VEL
LIN {X 0,Y 608.452,Z 170.757,A -85,B 0,C 180,E1 -460.314,E2 -460.314} C_VEL
LIN {X 0,Y 608.483,Z 152.921,A -85,B 0,C 180,E1 -463.186,E2 -463.186} C_VEL
LIN {X 0,Y 608.464,Z 135.134,A -85,B 0,C 180,E1 -466.094,E2 -466.094} C_VEL
LIN {X 0,Y 608.481,Z 119.291,A -85,B 0,C 180,E1 -468.719,E2 -468.719} C_VEL
LIN {X 0,Y 608.488,Z 107.561,A -85,B 0,C 180,E1 -470.725,E2 -470.725} C_VEL
LIN {X 0,Y 608.448,Z 107.502,A -85,B 0,C 180,E1 -473.124,E2 -473.124} C_VEL
LIN {X 0,Y 608.453,Z 107.501,A -85,B 0,C 180,E1 -475.717,E2 -475.717} C_VEL
LIN {X 0,Y 608.45,Z 107.509,A -85,B 0,C 180,E1 -478.267,E2 -478.267} C_VEL
LIN {X 0,Y 608.472,Z 107.504,A -85,B 0,C 180,E1 -480.545,E2 -480.545} C_VEL
LIN {X 0,Y 608.452,Z 107.502,A -85,B 0,C 180,E1 -482.88,E2 -482.88} C_VEL
LIN {X 0,Y 608.435,Z 107.503,A -85,B 0,C 180,E1 -485.278,E2 -485.278} C_VEL
LIN {X 0,Y 608.468,Z 107.505,A -85,B 0,C 180,E1 -488.24,E2 -488.24} C_VEL
LIN {X 0,Y 608.436,Z 107.503,A -85,B 0,C 180,E1 -491.178,E2 -491.178} C_VEL
LIN {X 0,Y 608.47,Z 107.507,A -85,B 0,C 180,E1 -493.869,E2 -493.869} C_VEL
LIN {X 0,Y 608.464,Z 107.499,A -85,B 0,C 180,E1 -496.692,E2 -496.692} C_VEL
LIN {X 0,Y 608.44,Z 107.502,A -85,B 0,C 180,E1 -498.822,E2 -498.822} C_VEL
LIN {X 0,Y 608.466,Z 107.505,A -85,B 0,C 180,E1 -501.76,E2 -501.76} C_VEL
LIN {X 0,Y 608.439,Z 107.503,A -85,B 0,C 180,E1 -504.722,E2 -504.722} C_VEL
LIN {X 0,Y 608.462,Z 107.506,A -85,B 0,C 180,E1 -507.478,E2 -507.478} C_VEL
LIN {X 0,Y 608.467,Z 107.498,A -85,B 0,C 180,E1 -510.22,E2 -510.22} C_VEL
LIN {X 0,Y 608.475,Z 107.503,A -85,B 0,C 180,E1 -512.794,E2 -512.794} C_VEL
LIN {X 0,Y 608.479,Z 107.497,A -85,B 0,C 180,E1 -515.847,E2 -515.847} C_VEL
LIN {X 0,Y 608.463,Z 107.501,A -85,B 0,C 180,E1 -518.308,E2 -518.308} C_VEL
LIN {X 0,Y 608.472,Z 107.5,A -85,B 0,C 180,E1 -521.284,E2 -521.284} C_VEL
LIN {X 0,Y 608.453,Z 107.501,A -85,B 0,C 180,E1 -523.906,E2 -523.906} C_VEL
LIN {X 0,Y 608.462,Z 107.508,A -85,B 0,C 180,E1 -526.644,E2 -526.644} C_VEL
LIN {X 0,Y 608.464,Z 107.499,A -85,B 0,C 180,E1 -529.35,E2 -529.35} C_VEL
LIN {X 0,Y 608.475,Z 107.502,A -85,B 0,C 180,E1 -532.033,E2 -532.033} C_VEL
LIN {X 0,Y 608.462,Z 107.503,A -85,B 0,C 180,E1 -534.698,E2 -534.698} C_VEL
LIN {X 0,Y 608.472,Z 107.498,A -85,B 0,C 180,E1 -537.352,E2 -537.352} C_VEL
LIN {X 0,Y 608.477,Z 107.506,A -85,B 0,C 180,E1 -540,E2 -540} C_VEL
LIN {X 0,Y 608.473,Z 107.499,A -85,B 0,C 180,E1 -542.648,E2 -542.648} C_VEL
LIN {X 0,Y 608.457,Z 107.502,A -85,B 0,C 180,E1 -545.302,E2 -545.302} C_VEL
LIN {X 0,Y 608.479,Z 107.504,A -85,B 0,C 180,E1 -547.967,E2 -547.967} C_VEL
LIN {X 0,Y 608.455,Z 107.503,A -85,B 0,C 180,E1 -549.455,E2 -549.455} C_VEL
LIN {X 0,Y 607.781,Z 107.59,A -85,B 0,C 180,E1 -550.008,E2 -550.008} C_VEL
LIN {X 0,Y 604.929,Z 107.943,A -85,B 0,C 180,E1 -550.905,E2 -550.905} C_VEL
LIN {X 0,Y 602.525,Z 108.249,A -85,B 0,C 180,E1 -551.626,E2 -551.626} C_VEL
LIN {X 0,Y 601.494,Z 108.37,A -85,B 0,C 180,E1 -552.183,E2 -552.183} C_VEL
LIN {X 0,Y 601.41,Z 108.378,A -85,B 0,C 180,E1 -552.371,E2 -552.371} C_VEL
LIN {X 0,Y 601.431,Z 108.377,A -85,B 0,C 180,E1 -554.897,E2 -554.897} C_VEL
LIN {X 0,Y 601.433,Z 108.378,A -85,B 0,C 180,E1 -556.986,E2 -556.986} C_VEL
LIN {X 0,Y 601.405,Z 108.381,A -85,B 0,C 180,E1 -559.81,E2 -559.81} C_VEL
LIN {X 0,Y 601.413,Z 108.379,A -85,B 0,C 180,E1 -562.683,E2 -562.683} C_VEL
LIN {X 0,Y 601.403,Z 108.384,A -85,B 0,C 180,E1 -564.879,E2 -564.879} C_VEL
LIN {X 0,Y 601.42,Z 108.381,A -85,B 0,C 180,E1 -567.363,E2 -567.363} C_VEL
LIN {X 0,Y 601.43,Z 108.376,A -85,B 0,C 180,E1 -570.164,E2 -570.164} C_VEL
LIN {X 0,Y 601.418,Z 108.385,A -85,B 0,C 180,E1 -572.715,E2 -572.715} C_VEL
LIN {X 0,Y 601.403,Z 108.383,A -85,B 0,C 180,E1 -575.113,E2 -575.113} C_VEL
LIN {X 0,Y 601.434,Z 108.375,A -85,B 0,C 180,E1 -577.419,E2 -577.419} C_VEL
LIN {X 0,Y 601.404,Z 108.38,A -85,B 0,C 180,E1 -579.996,E2 -579.996} C_VEL
LIN {X 0,Y 601.41,Z 108.384,A -85,B 0,C 180,E1 -582.671,E2 -582.671} C_VEL
LIN {X 0,Y 601.4,Z 108.379,A -85,B 0,C 180,E1 -585.479,E2 -585.479} C_VEL
LIN {X 0,Y 601.42,Z 108.384,A -85,B 0,C 180,E1 -588.407,E2 -588.407} C_VEL
LIN {X 0,Y 601.41,Z 108.378,A -85,B 0,C 180,E1 -590.873,E2 -590.873} C_VEL
LIN {X 0,Y 601.406,Z 108.379,A -85,B 0,C 180,E1 -593.417,E2 -593.417} C_VEL
LIN {X 0,Y 601.419,Z 108.385,A -85,B 0,C 180,E1 -596.066,E2 -596.066} C_VEL
LIN {X 0,Y 601.419,Z 108.378,A -85,B 0,C 180,E1 -598.546,E2 -598.546} C_VEL
LIN {X 0,Y 601.432,Z 108.379,A -85,B 0,C 180,E1 -601.373,E2 -601.373} C_VEL
LIN {X 0,Y 601.404,Z 108.388,A -85,B 0,C 180,E1 -603.636,E2 -603.636} C_VEL
LIN {X 0,Y 601.45,Z 108.378,A -85,B 0,C 180,E1 -605.859,E2 -605.859} C_VEL
LIN {X 0,Y 601.406,Z 108.379,A -85,B 0,C 180,E1 -608.761,E2 -608.761} C_VEL
LIN {X 0,Y 601.484,Z 108.566,A -85,B 0,C 180,E1 -611.364,E2 -611.364} C_VEL
LIN {X 0,Y 601.421,Z 122.453,A -85,B 0,C 180,E1 -614.061,E2 -614.061} C_VEL
LIN {X 0,Y 601.402,Z 136.941,A -85,B 0,C 180,E1 -616.828,E2 -616.828} C_VEL
LIN {X 0,Y 601.405,Z 151.999,A -85,B 0,C 180,E1 -619.649,E2 -619.649} C_VEL
LIN {X 0,Y 601.518,Z 153.318,A -85,B 0,C 180,E1 -619.715,E2 -619.715} C_VEL
LIN {X 0,Y 601.506,Z 228.279,A -85,B 0,C 180,E1 -620.628,E2 -620.628} C_VEL
LIN {X 0,Y 601.488,Z 238.803,A -85,B 0,C 180,E1 -620.861,E2 -620.861} C_VEL
LIN {X 0,Y 601.473,Z 250.536,A -85,B 0,C 180,E1 -621.263,E2 -621.263} C_VEL
LIN {X 0,Y 601.455,Z 260.931,A -85,B 0,C 180,E1 -621.77,E2 -621.77} C_VEL
LIN {X 0,Y 601.437,Z 269.114,A -85,B 0,C 180,E1 -622.277,E2 -622.277} C_VEL
LIN {X 0,Y 601.414,Z 276.875,A -85,B 0,C 180,E1 -622.868,E2 -622.868} C_VEL
LIN {X 0,Y 601.394,Z 284.708,A -85,B 0,C 180,E1 -623.598,E2 -623.598} C_VEL
LIN {X 0,Y 601.383,Z 292.114,A -85,B 0,C 180,E1 -624.467,E2 -624.467} C_VEL
LIN {X 0,Y 601.34,Z 297.728,A -85,B 0,C 180,E1 -625.307,E2 -625.307} C_VEL
LIN {X 0,Y 601.366,Z 302.943,A -85,B 0,C 180,E1 -626.315,E2 -626.315} C_VEL
LIN {X 0,Y 601.345,Z 305.633,A -85,B 0,C 180,E1 -626.985,E2 -626.985} C_VEL
LIN {X 0,Y 601.342,Z 308.572,A -85,B 0,C 180,E1 -627.991,E2 -627.991} C_VEL
LIN {X 0,Y 601.345,Z 309.871,A -85,B 0,C 180,E1 -628.66,E2 -628.66} C_VEL
LIN {X 0,Y 601.335,Z 310.692,A -85,B 0,C 180,E1 -629.33,E2 -629.33} C_VEL
LIN {X 0,Y 601.333,Z 310.996,A -85,B 0,C 180,E1 -630,E2 -630} C_VEL
LIN {X 0,Y 601.336,Z 310.735,A -85,B 0,C 180,E1 -630.669,E2 -630.669} C_VEL
LIN {X 0,Y 601.346,Z 309.998,A -85,B 0,C 180,E1 -631.339,E2 -631.339} C_VEL
LIN {X 0,Y 601.342,Z 308.788,A -85,B 0,C 180,E1 -632.009,E2 -632.009} C_VEL
LIN {X 0,Y 601.344,Z 305.942,A -85,B 0,C 180,E1 -633.015,E2 -633.015} C_VEL
LIN {X 0,Y 601.365,Z 303.351,A -85,B 0,C 180,E1 -633.685,E2 -633.685} C_VEL
LIN {X 0,Y 601.362,Z 298.243,A -85,B 0,C 180,E1 -634.692,E2 -634.692} C_VEL
LIN {X 0,Y 601.384,Z 292.747,A -85,B 0,C 180,E1 -635.532,E2 -635.532} C_VEL
LIN {X 0,Y 601.394,Z 284.589,A -85,B 0,C 180,E1 -636.504,E2 -636.504} C_VEL
LIN {X 0,Y 601.414,Z 276.947,A -85,B 0,C 180,E1 -637.217,E2 -637.217} C_VEL
LIN {X 0,Y 601.416,Z 269.198,A -85,B 0,C 180,E1 -637.807,E2 -637.807} C_VEL
LIN {X 0,Y 601.447,Z 261.033,A -85,B 0,C 180,E1 -638.314,E2 -638.314} C_VEL
LIN {X 0,Y 601.461,Z 250.662,A -85,B 0,C 180,E1 -638.822,E2 -638.822} C_VEL
LIN {X 0,Y 601.493,Z 239.021,A -85,B 0,C 180,E1 -639.224,E2 -639.224} C_VEL
LIN {X 0,Y 601.518,Z 228.616,A -85,B 0,C 180,E1 -639.457,E2 -639.457} C_VEL
LIN {X 0,Y 601.553,Z 180.357,A -85,B 0,C 180,E1 -640.05,E2 -640.05} C_VEL
LIN {X 0,Y 601.44,Z 152.687,A -85,B 0,C 180,E1 -640.392,E2 -640.392} C_VEL
LIN {X 0,Y 601.384,Z 151.478,A -85,B 0,C 180,E1 -640.521,E2 -640.521} C_VEL
LIN {X 0,Y 601.4,Z 137.417,A -85,B 0,C 180,E1 -643.172,E2 -643.172} C_VEL
LIN {X 0,Y 601.418,Z 124.734,A -85,B 0,C 180,E1 -645.591,E2 -645.591} C_VEL
LIN {X 0,Y 601.484,Z 110.239,A -85,B 0,C 180,E1 -648.39,E2 -648.39} C_VEL
LIN {X 0,Y 601.428,Z 108.436,A -85,B 0,C 180,E1 -648.778,E2 -648.778} C_VEL
LIN {X 0,Y 601.406,Z 108.38,A -85,B 0,C 180,E1 -651.239,E2 -651.239} C_VEL
LIN {X 0,Y 601.444,Z 108.378,A -85,B 0,C 180,E1 -654.141,E2 -654.141} C_VEL
LIN {X 0,Y 601.455,Z 108.373,A -85,B 0,C 180,E1 -657.111,E2 -657.111} C_VEL
LIN {X 0,Y 601.41,Z 108.378,A -85,B 0,C 180,E1 -659.393,E2 -659.393} C_VEL
LIN {X 0,Y 601.4,Z 108.382,A -85,B 0,C 180,E1 -661.727,E2 -661.727} C_VEL
LIN {X 0,Y 601.422,Z 108.387,A -85,B 0,C 180,E1 -664.118,E2 -664.118} C_VEL
LIN {X 0,Y 601.405,Z 108.38,A -85,B 0,C 180,E1 -666.583,E2 -666.583} C_VEL
LIN {X 0,Y 601.408,Z 108.378,A -85,B 0,C 180,E1 -669.126,E2 -669.126} C_VEL
LIN {X 0,Y 601.422,Z 108.386,A -85,B 0,C 180,E1 -671.765,E2 -671.765} C_VEL
LIN {X 0,Y 601.396,Z 108.38,A -85,B 0,C 180,E1 -674.532,E2 -674.532} C_VEL
LIN {X 0,Y 601.413,Z 108.384,A -85,B 0,C 180,E1 -677.409,E2 -677.409} C_VEL
LIN {X 0,Y 601.402,Z 108.381,A -85,B 0,C 180,E1 -680.004,E2 -680.004} C_VEL
LIN {X 0,Y 601.432,Z 108.375,A -85,B 0,C 180,E1 -682.618,E2 -682.618} C_VEL
LIN {X 0,Y 601.414,Z 108.383,A -85,B 0,C 180,E1 -685.068,E2 -685.068} C_VEL
LIN {X 0,Y 601.428,Z 108.381,A -85,B 0,C 180,E1 -687.484,E2 -687.484} C_VEL
LIN {X 0,Y 601.428,Z 108.376,A -85,B 0,C 180,E1 -689.851,E2 -689.851} C_VEL
LIN {X 0,Y 601.417,Z 108.381,A -85,B 0,C 180,E1 -692.637,E2 -692.637} C_VEL
LIN {X 0,Y 601.403,Z 108.385,A -85,B 0,C 180,E1 -695.121,E2 -695.121} C_VEL
LIN {X 0,Y 601.414,Z 108.379,A -85,B 0,C 180,E1 -697.394,E2 -697.394} C_VEL
LIN {X 0,Y 601.405,Z 108.38,A -85,B 0,C 180,E1 -700.19,E2 -700.19} C_VEL
LIN {X 0,Y 601.433,Z 108.379,A -85,B 0,C 180,E1 -703.014,E2 -703.014} C_VEL
LIN {X 0,Y 601.42,Z 108.378,A -85,B 0,C 180,E1 -705.908,E2 -705.908} C_VEL
LIN {X 0,Y 601.432,Z 108.383,A -85,B 0,C 180,E1 -708.542,E2 -708.542} C_VEL
LIN {X 0,Y 601.415,Z 108.377,A -85,B 0,C 180,E1 -711.262,E2 -711.262} C_VEL
LIN {X 0,Y 601.417,Z 108.383,A -85,B 0,C 180,E1 -713.963,E2 -713.963} C_VEL
LIN {X 0,Y 601.422,Z 108.378,A -85,B 0,C 180,E1 -716.65,E2 -716.65} C_VEL
LIN {X 0,Y 601.448,Z 108.374,A -85,B 0,C 180,E1 -719.33,E2 -719.33} C_VEL
LIN {X 0,Y 601.433,Z 108.383,A -85,B 0,C 180,E1 -722.009,E2 -722.009} C_VEL
LIN {X 0,Y 601.42,Z 108.377,A -85,B 0,C 180,E1 -724.692,E2 -724.692} C_VEL
LIN {X 0,Y 601.438,Z 108.379,A -85,B 0,C 180,E1 -727.385,E2 -727.385} C_VEL
LIN {X 0,Y 601.431,Z 108.378,A -85,B 0,C 180,E1 -730.095,E2 -730.095} C_VEL
LIN {X 0,Y 601.422,Z 108.377,A -85,B 0,C 180,E1 -732.828,E2 -732.828} C_VEL
LIN {X 0,Y 601.411,Z 108.384,A -85,B 0,C 180,E1 -735.591,E2 -735.591} C_VEL
LIN {X 0,Y 601.416,Z 108.377,A -85,B 0,C 180,E1 -738.392,E2 -738.392} C_VEL
LIN {X 0,Y 601.404,Z 108.387,A -85,B 0,C 180,E1 -741.239,E2 -741.239} C_VEL
LIN {X 0,Y 601.457,Z 108.372,A -85,B 0,C 180,E1 -744.14,E2 -744.14} C_VEL
LIN {X 0,Y 601.447,Z 108.38,A -85,B 0,C 180,E1 -747.111,E2 -747.111} C_VEL
LIN {X 0,Y 601.416,Z 108.379,A -85,B 0,C 180,E1 -749.393,E2 -749.393} C_VEL
LIN {X 0,Y 601.399,Z 108.379,A -85,B 0,C 180,E1 -751.727,E2 -751.727} C_VEL
LIN {X 0,Y 601.429,Z 108.377,A -85,B 0,C 180,E1 -754.118,E2 -754.118} C_VEL
LIN {X 0,Y 601.406,Z 108.388,A -85,B 0,C 180,E1 -756.583,E2 -756.583} C_VEL
LIN {X 0,Y 601.408,Z 108.379,A -85,B 0,C 180,E1 -759.127,E2 -759.127} C_VEL
LIN {X 0,Y 601.423,Z 108.378,A -85,B 0,C 180,E1 -761.765,E2 -761.765} C_VEL
LIN {X 0,Y 601.423,Z 108.382,A -85,B 0,C 180,E1 -764.535,E2 -764.535} C_VEL
LIN {X 0,Y 601.41,Z 108.378,A -85,B 0,C 180,E1 -767.409,E2 -767.409} C_VEL
LIN {X 0,Y 601.402,Z 108.388,A -85,B 0,C 180,E1 -770.005,E2 -770.005} C_VEL
LIN {X 0,Y 601.431,Z 108.376,A -85,B 0,C 180,E1 -772.618,E2 -772.618} C_VEL
LIN {X 0,Y 601.439,Z 108.374,A -85,B 0,C 180,E1 -775.07,E2 -775.07} C_VEL
LIN {X 0,Y 601.434,Z 108.38,A -85,B 0,C 180,E1 -777.485,E2 -777.485} C_VEL
LIN {X 0,Y 601.426,Z 108.383,A -85,B 0,C 180,E1 -779.852,E2 -779.852} C_VEL
LIN {X 0,Y 601.414,Z 108.377,A -85,B 0,C 180,E1 -782.638,E2 -782.638} C_VEL
LIN {X 0,Y 601.398,Z 108.383,A -85,B 0,C 180,E1 -785.121,E2 -785.121} C_VEL
LIN {X 0,Y 601.403,Z 108.382,A -85,B 0,C 180,E1 -788.041,E2 -788.041} C_VEL
LIN {X 0,Y 601.451,Z 108.499,A -85,B 0,C 180,E1 -789.197,E2 -789.197} C_VEL
LIN {X 0,Y 601.504,Z 119.889,A -85,B 0,C 180,E1 -791.157,E2 -791.157} C_VEL
LIN {X 0,Y 601.443,Z 136.182,A -85,B 0,C 180,E1 -793.888,E2 -793.888} C_VEL
LIN {X 0,Y 601.44,Z 152.923,A -85,B 0,C 180,E1 -796.657,E2 -796.657} C_VEL
LIN {X 0,Y 601.378,Z 169.664,A -85,B 0,C 180,E1 -799.394,E2 -799.394} C_VEL
LIN {X 0,Y 601.425,Z 171.415,A -85,B 0,C 180,E1 -799.629,E2 -799.629} C_VEL
LIN {X 0,Y 601.531,Z 180.469,A -85,B 0,C 180,E1 -799.758,E2 -799.758} C_VEL
LIN {X 0,Y 601.524,Z 248.453,A -85,B 0,C 180,E1 -800.586,E2 -800.586} C_VEL
LIN {X 0,Y 601.51,Z 258.912,A -85,B 0,C 180,E1 -800.819,E2 -800.819} C_VEL
LIN {X 0,Y 601.472,Z 269.62,A -85,B 0,C 180,E1 -801.178,E2 -801.178} C_VEL
LIN {X 0,Y 601.446,Z 280.24,A -85,B 0,C 180,E1 -801.686,E2 -801.686} C_VEL
LIN {X 0,Y 601.416,Z 288.547,A -85,B 0,C 180,E1 -802.193,E2 -802.193} C_VEL
LIN {X 0,Y 601.412,Z 296.404,A -85,B 0,C 180,E1 -802.783,E2 -802.783} C_VEL
LIN {X 0,Y 601.411,Z 303.598,A -85,B 0,C 180,E1 -803.443,E2 -803.443} C_VEL
LIN {X 0,Y 601.391,Z 311.192,A -85,B 0,C 180,E1 -804.299,E2 -804.299} C_VEL
LIN {X 0,Y 601.38,Z 317.029,A -85,B 0,C 180,E1 -805.14,E2 -805.14} C_VEL
LIN {X 0,Y 601.345,Z 321.632,A -85,B 0,C 180,E1 -805.979,E2 -805.979} C_VEL
LIN {X 0,Y 601.343,Z 324.622,A -85,B 0,C 180,E1 -806.65,E2 -806.65} C_VEL
LIN {X 0,Y 601.326,Z 326.932,A -85,B 0,C 180,E1 -807.321,E2 -807.321} C_VEL
LIN {X 0,Y 601.342,Z 328.679,A -85,B 0,C 180,E1 -807.991,E2 -807.991} C_VEL
LIN {X 0,Y 601.345,Z 329.935,A -85,B 0,C 180,E1 -808.661,E2 -808.661} C_VEL
LIN {X 0,Y 601.335,Z 330.713,A -85,B 0,C 180,E1 -809.331,E2 -809.331} C_VEL
LIN {X 0,Y 601.332,Z 331,A -85,B 0,C 180,E1 -810,E2 -810} C_VEL
LIN {X 0,Y 601.335,Z 330.713,A -85,B 0,C 180,E1 -810.67,E2 -810.67} C_VEL
LIN {X 0,Y 601.345,Z 329.934,A -85,B 0,C 180,E1 -811.34,E2 -811.34} C_VEL
LIN {X 0,Y 601.342,Z 328.678,A -85,B 0,C 180,E1 -812.009,E2 -812.009} C_VEL
LIN {X 0,Y 601.342,Z 325.786,A -85,B 0,C 180,E1 -813.015,E2 -813.015} C_VEL
LIN {X 0,Y 601.364,Z 323.146,A -85,B 0,C 180,E1 -813.686,E2 -813.686} C_VEL
LIN {X 0,Y 601.341,Z 317.984,A -85,B 0,C 180,E1 -814.693,E2 -814.693} C_VEL
LIN {X 0,Y 601.383,Z 312.429,A -85,B 0,C 180,E1 -815.533,E2 -815.533} C_VEL
LIN {X 0,Y 601.393,Z 305.151,A -85,B 0,C 180,E1 -816.403,E2 -816.403} C_VEL
LIN {X 0,Y 601.415,Z 297.415,A -85,B 0,C 180,E1 -817.132,E2 -817.132} C_VEL
LIN {X 0,Y 601.436,Z 289.761,A -85,B 0,C 180,E1 -817.723,E2 -817.723} C_VEL
LIN {X 0,Y 601.454,Z 281.721,A -85,B 0,C 180,E1 -818.23,E2 -818.23} C_VEL
LIN {X 0,Y 601.481,Z 273.39,A -85,B 0,C 180,E1 -818.652,E2 -818.652} C_VEL
LIN {X 0,Y 601.471,Z 264.886,A -85,B 0,C 180,E1 -818.991,E2 -818.991} C_VEL
LIN {X 0,Y 601.498,Z 255.579,A -85,B 0,C 180,E1 -819.266,E2 -819.266} C_VEL
LIN {X 0,Y 601.533,Z 244.538,A -85,B 0,C 180,E1 -819.478,E2 -819.478} C_VEL
LIN {X 0,Y 601.455,Z 171.923,A -85,B 0,C 180,E1 -820.35,E2 -820.35} C_VEL
LIN {X 0,Y 601.39,Z 170.757,A -85,B 0,C 180,E1 -820.436,E2 -820.436} C_VEL
LIN {X 0,Y 601.423,Z 153.967,A -85,B 0,C 180,E1 -823.172,E2 -823.172} C_VEL
LIN {X 0,Y 601.466,Z 137.227,A -85,B 0,C 180,E1 -825.938,E2 -825.938} C_VEL
LIN {X 0,Y 601.498,Z 121.233,A -85,B 0,C 180,E1 -828.616,E2 -828.616} C_VEL
LIN {X 0,Y 601.452,Z 108.576,A -85,B 0,C 180,E1 -830.777,E2 -830.777} C_VEL
LIN {X 0,Y 601.391,Z 108.376,A -85,B 0,C 180,E1 -833.412,E2 -833.412} C_VEL
LIN {X 0,Y 601.397,Z 108.381,A -85,B 0,C 180,E1 -835.864,E2 -835.864} C_VEL
LIN {X 0,Y 601.401,Z 108.381,A -85,B 0,C 180,E1 -837.868,E2 -837.868} C_VEL
LIN {X 0,Y 601.428,Z 108.383,A -85,B 0,C 180,E1 -840.164,E2 -840.164} C_VEL
LIN {X 0,Y 601.422,Z 108.379,A -85,B 0,C 180,E1 -842.715,E2 -842.715} C_VEL
LIN {X 0,Y 601.398,Z 108.379,A -85,B 0,C 180,E1 -845.112,E2 -845.112} C_VEL
LIN {X 0,Y 601.432,Z 108.376,A -85,B 0,C 180,E1 -847.419,E2 -847.419} C_VEL
LIN {X 0,Y 601.402,Z 108.388,A -85,B 0,C 180,E1 -849.996,E2 -849.996} C_VEL
LIN {X 0,Y 601.408,Z 108.378,A -85,B 0,C 180,E1 -852.671,E2 -852.671} C_VEL
LIN {X 0,Y 601.399,Z 108.385,A -85,B 0,C 180,E1 -855.48,E2 -855.48} C_VEL
LIN {X 0,Y 601.421,Z 108.377,A -85,B 0,C 180,E1 -858.407,E2 -858.407} C_VEL
LIN {X 0,Y 601.407,Z 108.379,A -85,B 0,C 180,E1 -860.873,E2 -860.873} C_VEL
LIN {X 0,Y 601.443,Z 108.379,A -85,B 0,C 180,E1 -863.734,E2 -863.734} C_VEL
LIN {X 0,Y 601.414,Z 108.378,A -85,B 0,C 180,E1 -866.686,E2 -866.686} C_VEL
LIN {X 0,Y 601.414,Z 108.384,A -85,B 0,C 180,E1 -869.058,E2 -869.058} C_VEL
LIN {X 0,Y 601.433,Z 108.381,A -85,B 0,C 180,E1 -871.373,E2 -871.373} C_VEL
LIN {X 0,Y 601.4,Z 108.381,A -85,B 0,C 180,E1 -873.636,E2 -873.636} C_VEL
LIN {X 0,Y 601.457,Z 108.372,A -85,B 0,C 180,E1 -875.86,E2 -875.86} C_VEL
LIN {X 0,Y 601.404,Z 108.387,A -85,B 0,C 180,E1 -878.761,E2 -878.761} C_VEL
LIN {X 0,Y 601.401,Z 108.379,A -85,B 0,C 180,E1 -881.608,E2 -881.608} C_VEL
LIN {X 0,Y 601.436,Z 108.374,A -85,B 0,C 180,E1 -883.713,E2 -883.713} C_VEL
LIN {X 0,Y 601.412,Z 108.386,A -85,B 0,C 180,E1 -886.484,E2 -886.484} C_VEL
LIN {X 0,Y 601.419,Z 108.377,A -85,B 0,C 180,E1 -889.224,E2 -889.224} C_VEL
LIN {X 0,Y 601.439,Z 108.377,A -85,B 0,C 180,E1 -891.939,E2 -891.939} C_VEL
LIN {X 0,Y 601.426,Z 108.38,A -85,B 0,C 180,E1 -894.636,E2 -894.636} C_VEL
LIN {X 0,Y 601.438,Z 108.374,A -85,B 0,C 180,E1 -897.321,E2 -897.321} C_VEL
LIN {X 0,Y 601.446,Z 108.382,A -85,B 0,C 180,E1 -900,E2 -900} C_VEL
LIN {X 0,Y 601.439,Z 108.375,A -85,B 0,C 180,E1 -902.679,E2 -902.679} C_VEL
LIN {X 0,Y 601.423,Z 108.379,A -85,B 0,C 180,E1 -905.364,E2 -905.364} C_VEL
LIN {X 0,Y 601.442,Z 108.379,A -85,B 0,C 180,E1 -908.061,E2 -908.061} C_VEL
LIN {X 0,Y 601.427,Z 108.377,A -85,B 0,C 180,E1 -911.013,E2 -911.013} C_VEL
LIN {X 0,Y 601.41,Z 108.378,A -85,B 0,C 180,E1 -912.371,E2 -912.371} C_VEL
LIN {X 0,Y 600.745,Z 108.462,A -85,B 0,C 180,E1 -912.93,E2 -912.93} C_VEL
LIN {X 0,Y 597.896,Z 108.821,A -85,B 0,C 180,E1 -913.838,E2 -913.838} C_VEL
LIN {X 0,Y 595.486,Z 109.12,A -85,B 0,C 180,E1 -914.568,E2 -914.568} C_VEL
LIN {X 0,Y 594.447,Z 109.249,A -85,B 0,C 180,E1 -915.132,E2 -915.132} C_VEL
LIN {X 0,Y 594.361,Z 109.258,A -85,B 0,C 180,E1 -915.323,E2 -915.323} C_VEL
LIN {X 0,Y 594.391,Z 109.258,A -85,B 0,C 180,E1 -917.193,E2 -917.193} C_VEL
LIN {X 0,Y 594.374,Z 109.255,A -85,B 0,C 180,E1 -920.054,E2 -920.054} C_VEL
LIN {X 0,Y 594.358,Z 109.262,A -85,B 0,C 180,E1 -922.968,E2 -922.968} C_VEL
LIN {X 0,Y 594.374,Z 109.263,A -85,B 0,C 180,E1 -925.193,E2 -925.193} C_VEL
LIN {X 0,Y 594.388,Z 109.255,A -85,B 0,C 180,E1 -927.527,E2 -927.527} C_VEL
LIN {X 0,Y 594.388,Z 109.254,A -85,B 0,C 180,E1 -930.328,E2 -930.328} C_VEL
LIN {X 0,Y 594.377,Z 109.262,A -85,B 0,C 180,E1 -932.95,E2 -932.95} C_VEL
LIN {X 0,Y 594.359,Z 109.257,A -85,B 0,C 180,E1 -935.408,E2 -935.408} C_VEL
LIN {X 0,Y 594.385,Z 109.254,A -85,B 0,C 180,E1 -937.941,E2 -937.941} C_VEL
LIN {X 0,Y 594.374,Z 109.259,A -85,B 0,C 180,E1 -940.822,E2 -940.822} C_VEL
LIN {X 0,Y 594.367,Z 109.255,A -85,B 0,C 180,E1 -943.3,E2 -943.3} C_VEL
LIN {X 0,Y 594.361,Z 109.263,A -85,B 0,C 180,E1 -946.161,E2 -946.161} C_VEL
LIN {X 0,Y 594.378,Z 109.259,A -85,B 0,C 180,E1 -948.536,E2 -948.536} C_VEL
LIN {X 0,Y 594.382,Z 109.253,A -85,B 0,C 180,E1 -951.296,E2 -951.296} C_VEL
LIN {X 0,Y 594.363,Z 109.261,A -85,B 0,C 180,E1 -953.756,E2 -953.756} C_VEL
LIN {X 0,Y 594.366,Z 109.26,A -85,B 0,C 180,E1 -956.238,E2 -956.238} C_VEL
LIN {X 0,Y 594.37,Z 109.255,A -85,B 0,C 180,E1 -958.65,E2 -958.65} C_VEL
LIN {X 0,Y 594.384,Z 109.254,A -85,B 0,C 180,E1 -961.042,E2 -961.042} C_VEL
LIN {X 0,Y 594.388,Z 109.256,A -85,B 0,C 180,E1 -963.301,E2 -963.301} C_VEL
LIN {X 0,Y 594.373,Z 109.255,A -85,B 0,C 180,E1 -966.295,E2 -966.295} C_VEL
LIN {X 0,Y 594.406,Z 109.257,A -85,B 0,C 180,E1 -969.224,E2 -969.224} C_VEL
LIN {X 0,Y 594.431,Z 109.417,A -85,B 0,C 180,E1 -971.301,E2 -971.301} C_VEL
LIN {X 0,Y 594.402,Z 122.456,A -85,B 0,C 180,E1 -973.868,E2 -973.868} C_VEL
LIN {X 0,Y 594.367,Z 136.944,A -85,B 0,C 180,E1 -976.669,E2 -976.669} C_VEL
LIN {X 0,Y 594.315,Z 152,A -85,B 0,C 180,E1 -979.524,E2 -979.524} C_VEL
LIN {X 0,Y 594.469,Z 153.312,A -85,B 0,C 180,E1 -979.592,E2 -979.592} C_VEL
LIN {X 0,Y 594.521,Z 228.313,A -85,B 0,C 180,E1 -980.517,E2 -980.517} C_VEL
LIN {X 0,Y 594.487,Z 238.828,A -85,B 0,C 180,E1 -980.752,E2 -980.752} C_VEL
LIN {X 0,Y 594.458,Z 250.545,A -85,B 0,C 180,E1 -981.159,E2 -981.159} C_VEL
LIN {X 0,Y 594.431,Z 260.946,A -85,B 0,C 180,E1 -981.672,E2 -981.672} C_VEL
LIN {X 0,Y 594.373,Z 269.125,A -85,B 0,C 180,E1 -982.185,E2 -982.185} C_VEL
LIN {X 0,Y 594.356,Z 276.883,A -85,B 0,C 180,E1 -982.782,E2 -982.782} C_VEL
LIN {X 0,Y 594.345,Z 284.714,A -85,B 0,C 180,E1 -983.522,E2 -983.522} C_VEL
LIN {X 0,Y 594.309,Z 292.119,A -85,B 0,C 180,E1 -984.401,E2 -984.401} C_VEL
LIN {X 0,Y 594.255,Z 297.732,A -85,B 0,C 180,E1 -985.251,E2 -985.251} C_VEL
LIN {X 0,Y 594.287,Z 302.946,A -85,B 0,C 180,E1 -986.271,E2 -986.271} C_VEL
LIN {X 0,Y 594.248,Z 305.636,A -85,B 0,C 180,E1 -986.949,E2 -986.949} C_VEL
LIN {X 0,Y 594.242,Z 308.575,A -85,B 0,C 180,E1 -987.967,E2 -987.967} C_VEL
LIN {X 0,Y 594.244,Z 309.873,A -85,B 0,C 180,E1 -988.644,E2 -988.644} C_VEL
LIN {X 0,Y 594.235,Z 310.691,A -85,B 0,C 180,E1 -989.322,E2 -989.322} C_VEL
LIN {X 0,Y 594.234,Z 310.996,A -85,B 0,C 180,E1 -990,E2 -990} C_VEL
LIN {X 0,Y 594.236,Z 310.734,A -85,B 0,C 180,E1 -990.677,E2 -990.677} C_VEL
LIN {X 0,Y 594.246,Z 309.998,A -85,B 0,C 180,E1 -991.355,E2 -991.355} C_VEL
LIN {X 0,Y 594.241,Z 308.788,A -85,B 0,C 180,E1 -992.033,E2 -992.033} C_VEL
LIN {X 0,Y 594.247,Z 305.941,A -85,B 0,C 180,E1 -993.051,E2 -993.051} C_VEL
LIN {X 0,Y 594.286,Z 303.349,A -85,B 0,C 180,E1 -993.729,E2 -993.729} C_VEL
LIN {X 0,Y 594.265,Z 298.241,A -85,B 0,C 180,E1 -994.748,E2 -994.748} C_VEL
LIN {X 0,Y 594.31,Z 292.743,A -85,B 0,C 180,E1 -995.599,E2 -995.599} C_VEL
LIN {X 0,Y 594.342,Z 285.618,A -85,B 0,C 180,E1 -996.476,E2 -996.476} C_VEL
LIN {X 0,Y 594.355,Z 276.942,A -85,B 0,C 180,E1 -997.303,E2 -997.303} C_VEL
LIN {X 0,Y 594.38,Z 269.194,A -85,B 0,C 180,E1 -997.9,E2 -997.9} C_VEL
LIN {X 0,Y 594.42,Z 261.028,A -85,B 0,C 180,E1 -998.413,E2 -998.413} C_VEL
LIN {X 0,Y 594.46,Z 250.646,A -85,B 0,C 180,E1 -998.926,E2 -998.926} C_VEL
LIN {X 0,Y 594.494,Z 239.003,A -85,B 0,C 180,E1 -999.333,E2 -999.333} C_VEL
LIN {X 0,Y 594.536,Z 228.585,A -85,B 0,C 180,E1 -999.569,E2 -999.569} C_VEL
LIN {X 0,Y 594.577,Z 180.312,A -85,B 0,C 180,E1 -1000.169,E2 -1000.169} C_VEL
LIN {X 0,Y 594.401,Z 152.962,A -85,B 0,C 180,E1 -1000.506,E2 -1000.506} C_VEL
LIN {X 0,Y 594.304,Z 151.736,A -85,B 0,C 180,E1 -1000.605,E2 -1000.605} C_VEL
LIN {X 0,Y 594.364,Z 137.414,A -85,B 0,C 180,E1 -1003.331,E2 -1003.331} C_VEL
LIN {X 0,Y 594.398,Z 122.92,A -85,B 0,C 180,E1 -1006.132,E2 -1006.132} C_VEL
LIN {X 0,Y 594.41,Z 109.391,A -85,B 0,C 180,E1 -1008.797,E2 -1008.797} C_VEL
LIN {X 0,Y 594.363,Z 109.256,A -85,B 0,C 180,E1 -1011.503,E2 -1011.503} C_VEL
LIN {X 0,Y 594.389,Z 109.262,A -85,B 0,C 180,E1 -1014.446,E2 -1014.446} C_VEL
LIN {X 0,Y 594.387,Z 109.258,A -85,B 0,C 180,E1 -1016.699,E2 -1016.699} C_VEL
LIN {X 0,Y 594.381,Z 109.254,A -85,B 0,C 180,E1 -1018.998,E2 -1018.998} C_VEL
LIN {X 0,Y 594.376,Z 109.256,A -85,B 0,C 180,E1 -1021.642,E2 -1021.642} C_VEL
LIN {X 0,Y 594.394,Z 109.254,A -85,B 0,C 180,E1 -1024.579,E2 -1024.579} C_VEL
LIN {X 0,Y 594.388,Z 109.256,A -85,B 0,C 180,E1 -1027.608,E2 -1027.608} C_VEL
LIN {X 0,Y 594.369,Z 109.256,A -85,B 0,C 180,E1 -1030.567,E2 -1030.567} C_VEL
LIN {X 0,Y 594.365,Z 109.258,A -85,B 0,C 180,E1 -1033.299,E2 -1033.299} C_VEL
LIN {X 0,Y 594.367,Z 109.257,A -85,B 0,C 180,E1 -1036.16,E2 -1036.16} C_VEL
LIN {X 0,Y 594.378,Z 109.254,A -85,B 0,C 180,E1 -1038.536,E2 -1038.536} C_VEL
LIN {X 0,Y 594.38,Z 109.261,A -85,B 0,C 180,E1 -1041.296,E2 -1041.296} C_VEL
LIN {X 0,Y 594.394,Z 109.255,A -85,B 0,C 180,E1 -1043.758,E2 -1043.758} C_VEL
LIN {X 0,Y 594.375,Z 109.254,A -85,B 0,C 180,E1 -1046.238,E2 -1046.238} C_VEL
LIN {X 0,Y 594.369,Z 109.257,A -85,B 0,C 180,E1 -1048.65,E2 -1048.65} C_VEL
LIN {X 0,Y 594.382,Z 109.263,A -85,B 0,C 180,E1 -1051.042,E2 -1051.042} C_VEL
LIN {X 0,Y 594.38,Z 109.253,A -85,B 0,C 180,E1 -1053.978,E2 -1053.978} C_VEL
LIN {X 0,Y 594.388,Z 109.254,A -85,B 0,C 180,E1 -1056.296,E2 -1056.296} C_VEL
LIN {X 0,Y 594.403,Z 109.254,A -85,B 0,C 180,E1 -1059.224,E2 -1059.224} C_VEL
LIN {X 0,Y 594.353,Z 109.259,A -85,B 0,C 180,E1 -1062.095,E2 -1062.095} C_VEL
LIN {X 0,Y 594.364,Z 109.26,A -85,B 0,C 180,E1 -1064.219,E2 -1064.219} C_VEL
LIN {X 0,Y 594.379,Z 109.261,A -85,B 0,C 180,E1 -1066.321,E2 -1066.321} C_VEL
LIN {X 0,Y 594.377,Z 109.255,A -85,B 0,C 180,E1 -1069.095,E2 -1069.095} C_VEL
LIN {X 0,Y 594.413,Z 109.252,A -85,B 0,C 180,E1 -1071.843,E2 -1071.843} C_VEL
LIN {X 0,Y 594.39,Z 109.256,A -85,B 0,C 180,E1 -1074.572,E2 -1074.572} C_VEL
LIN {X 0,Y 594.405,Z 109.251,A -85,B 0,C 180,E1 -1077.289,E2 -1077.289} C_VEL
LIN {X 0,Y 594.414,Z 109.259,A -85,B 0,C 180,E1 -1080,E2 -1080} C_VEL
LIN {X 0,Y 594.404,Z 109.251,A -85,B 0,C 180,E1 -1082.711,E2 -1082.711} C_VEL
LIN {X 0,Y 594.39,Z 109.257,A -85,B 0,C 180,E1 -1085.428,E2 -1085.428} C_VEL
LIN {X 0,Y 594.413,Z 109.252,A -85,B 0,C 180,E1 -1088.157,E2 -1088.157} C_VEL
LIN {X 0,Y 594.39,Z 109.255,A -85,B 0,C 180,E1 -1091.075,E2 -1091.075} C_VEL
LIN {X 0,Y 594.38,Z 109.26,A -85,B 0,C 180,E1 -1093.679,E2 -1093.679} C_VEL
LIN {X 0,Y 594.395,Z 109.253,A -85,B 0,C 180,E1 -1096.72,E2 -1096.72} C_VEL
LIN {X 0,Y 594.367,Z 109.263,A -85,B 0,C 180,E1 -1099.334,E2 -1099.334} C_VEL
LIN {X 0,Y 594.364,Z 109.26,A -85,B 0,C 180,E1 -1101.503,E2 -1101.503} C_VEL
LIN {X 0,Y 594.388,Z 109.254,A -85,B 0,C 180,E1 -1104.446,E2 -1104.446} C_VEL
LIN {X 0,Y 594.382,Z 109.259,A -85,B 0,C 180,E1 -1106.7,E2 -1106.7} C_VEL
LIN {X 0,Y 594.38,Z 109.261,A -85,B 0,C 180,E1 -1108.998,E2 -1108.998} C_VEL
LIN {X 0,Y 594.375,Z 109.254,A -85,B 0,C 180,E1 -1111.643,E2 -1111.643} C_VEL
LIN {X 0,Y 594.381,Z 109.262,A -85,B 0,C 180,E1 -1114.58,E2 -1114.58} C_VEL
LIN {X 0,Y 594.381,Z 109.256,A -85,B 0,C 180,E1 -1117.087,E2 -1117.087} C_VEL
LIN {X 0,Y 594.358,Z 109.257,A -85,B 0,C 180,E1 -1119.773,E2 -1119.773} C_VEL
LIN {X 0,Y 594.369,Z 109.265,A -85,B 0,C 180,E1 -1122.375,E2 -1122.375} C_VEL
LIN {X 0,Y 594.342,Z 109.258,A -85,B 0,C 180,E1 -1125.193,E2 -1125.193} C_VEL
LIN {X 0,Y 594.367,Z 109.257,A -85,B 0,C 180,E1 -1127.625,E2 -1127.625} C_VEL
LIN {X 0,Y 594.369,Z 109.26,A -85,B 0,C 180,E1 -1130.319,E2 -1130.319} C_VEL
LIN {X 0,Y 594.38,Z 109.253,A -85,B 0,C 180,E1 -1132.913,E2 -1132.913} C_VEL
LIN {X 0,Y 594.375,Z 109.264,A -85,B 0,C 180,E1 -1135.862,E2 -1135.862} C_VEL
LIN {X 0,Y 594.367,Z 109.255,A -85,B 0,C 180,E1 -1138.65,E2 -1138.65} C_VEL
LIN {X 0,Y 594.383,Z 109.255,A -85,B 0,C 180,E1 -1141.042,E2 -1141.042} C_VEL
LIN {X 0,Y 594.386,Z 109.259,A -85,B 0,C 180,E1 -1143.301,E2 -1143.301} C_VEL
LIN {X 0,Y 594.368,Z 109.252,A -85,B 0,C 180,E1 -1146.295,E2 -1146.295} C_VEL
LIN {X 0,Y 594.444,Z 109.484,A -85,B 0,C 180,E1 -1149.121,E2 -1149.121} C_VEL
LIN {X 0,Y 594.535,Z 119.763,A -85,B 0,C 180,E1 -1150.906,E2 -1150.906} C_VEL
LIN {X 0,Y 594.437,Z 136.182,A -85,B 0,C 180,E1 -1153.693,E2 -1153.693} C_VEL
LIN {X 0,Y 594.412,Z 152.923,A -85,B 0,C 180,E1 -1156.496,E2 -1156.496} C_VEL
LIN {X 0,Y 594.322,Z 169.664,A -85,B 0,C 180,E1 -1159.266,E2 -1159.266} C_VEL
LIN {X 0,Y 594.362,Z 171.402,A -85,B 0,C 180,E1 -1159.504,E2 -1159.504} C_VEL
LIN {X 0,Y 594.545,Z 176.892,A -85,B 0,C 180,E1 -1159.593,E2 -1159.593} C_VEL
LIN {X 0,Y 594.54,Z 247.151,A -85,B 0,C 180,E1 -1160.453,E2 -1160.453} C_VEL
LIN {X 0,Y 594.509,Z 256.421,A -85,B 0,C 180,E1 -1160.645,E2 -1160.645} C_VEL
LIN {X 0,Y 594.462,Z 264.897,A -85,B 0,C 180,E1 -1160.902,E2 -1160.902} C_VEL
LIN {X 0,Y 594.446,Z 273.401,A -85,B 0,C 180,E1 -1161.245,E2 -1161.245} C_VEL
LIN {X 0,Y 594.431,Z 281.73,A -85,B 0,C 180,E1 -1161.673,E2 -1161.673} C_VEL
LIN {X 0,Y 594.372,Z 289.767,A -85,B 0,C 180,E1 -1162.185,E2 -1162.185} C_VEL
LIN {X 0,Y 594.356,Z 297.418,A -85,B 0,C 180,E1 -1162.783,E2 -1162.783} C_VEL
LIN {X 0,Y 594.33,Z 305.809,A -85,B 0,C 180,E1 -1163.589,E2 -1163.589} C_VEL
LIN {X 0,Y 594.309,Z 312.433,A -85,B 0,C 180,E1 -1164.401,E2 -1164.401} C_VEL
LIN {X 0,Y 594.256,Z 317.987,A -85,B 0,C 180,E1 -1165.251,E2 -1165.251} C_VEL
LIN {X 0,Y 594.286,Z 323.148,A -85,B 0,C 180,E1 -1166.271,E2 -1166.271} C_VEL
LIN {X 0,Y 594.245,Z 325.788,A -85,B 0,C 180,E1 -1166.949,E2 -1166.949} C_VEL
LIN {X 0,Y 594.241,Z 328.68,A -85,B 0,C 180,E1 -1167.967,E2 -1167.967} C_VEL
LIN {X 0,Y 594.245,Z 329.936,A -85,B 0,C 180,E1 -1168.645,E2 -1168.645} C_VEL
LIN {X 0,Y 594.235,Z 330.712,A -85,B 0,C 180,E1 -1169.323,E2 -1169.323} C_VEL
LIN {X 0,Y 594.233,Z 331,A -85,B 0,C 180,E1 -1170,E2 -1170} C_VEL
LIN {X 0,Y 594.235,Z 330.712,A -85,B 0,C 180,E1 -1170.678,E2 -1170.678} C_VEL
LIN {X 0,Y 594.245,Z 329.935,A -85,B 0,C 180,E1 -1171.356,E2 -1171.356} C_VEL
LIN {X 0,Y 594.241,Z 328.679,A -85,B 0,C 180,E1 -1172.033,E2 -1172.033} C_VEL
LIN {X 0,Y 594.245,Z 325.787,A -85,B 0,C 180,E1 -1173.051,E2 -1173.051} C_VEL
LIN {X 0,Y 594.286,Z 323.146,A -85,B 0,C 180,E1 -1173.729,E2 -1173.729} C_VEL
LIN {X 0,Y 594.256,Z 317.984,A -85,B 0,C 180,E1 -1174.749,E2 -1174.749} C_VEL
LIN {X 0,Y 594.319,Z 311.187,A -85,B 0,C 180,E1 -1175.769,E2 -1175.769} C_VEL
LIN {X 0,Y 594.342,Z 303.513,A -85,B 0,C 180,E1 -1176.644,E2 -1176.644} C_VEL
LIN {X 0,Y 594.354,Z 296.403,A -85,B 0,C 180,E1 -1177.303,E2 -1177.303} C_VEL
LIN {X 0,Y 594.375,Z 288.547,A -85,B 0,C 180,E1 -1177.901,E2 -1177.901} C_VEL
LIN {X 0,Y 594.445,Z 278.733,A -85,B 0,C 180,E1 -1178.499,E2 -1178.499} C_VEL
LIN {X 0,Y 594.467,Z 267.295,A -85,B 0,C 180,E1 -1179.012,E2 -1179.012} C_VEL
LIN {X 0,Y 594.518,Z 257.24,A -85,B 0,C 180,E1 -1179.333,E2 -1179.333} C_VEL
LIN {X 0,Y 594.536,Z 248.436,A -85,B 0,C 180,E1 -1179.526,E2 -1179.526} C_VEL
LIN {X 0,Y 594.554,Z 182.23,A -85,B 0,C 180,E1 -1180.342,E2 -1180.342} C_VEL
LIN {X 0,Y 594.395,Z 171.902,A -85,B 0,C 180,E1 -1180.474,E2 -1180.474} C_VEL
LIN {X 0,Y 594.317,Z 170.757,A -85,B 0,C 180,E1 -1180.562,E2 -1180.562} C_VEL
LIN {X 0,Y 594.391,Z 153.967,A -85,B 0,C 180,E1 -1183.33,E2 -1183.33} C_VEL
LIN {X 0,Y 594.435,Z 137.227,A -85,B 0,C 180,E1 -1186.131,E2 -1186.131} C_VEL
LIN {X 0,Y 594.502,Z 121.128,A -85,B 0,C 180,E1 -1188.862,E2 -1188.862} C_VEL
LIN {X 0,Y 594.461,Z 109.698,A -85,B 0,C 180,E1 -1190.833,E2 -1190.833} C_VEL
LIN {X 0,Y 594.386,Z 109.274,A -85,B 0,C 180,E1 -1191.002,E2 -1191.002} C_VEL
LIN {X 0,Y 594.368,Z 109.249,A -85,B 0,C 180,E1 -1193.705,E2 -1193.705} C_VEL
LIN {X 0,Y 594.386,Z 109.259,A -85,B 0,C 180,E1 -1196.7,E2 -1196.7} C_VEL
LIN {X 0,Y 594.382,Z 109.255,A -85,B 0,C 180,E1 -1198.999,E2 -1198.999} C_VEL
LIN {X 0,Y 594.376,Z 109.255,A -85,B 0,C 180,E1 -1201.642,E2 -1201.642} C_VEL
LIN {X 0,Y 594.382,Z 109.257,A -85,B 0,C 180,E1 -1204.58,E2 -1204.58} C_VEL
LIN {X 0,Y 594.388,Z 109.256,A -85,B 0,C 180,E1 -1207.608,E2 -1207.608} C_VEL
LIN {X 0,Y 594.37,Z 109.256,A -85,B 0,C 180,E1 -1210.567,E2 -1210.567} C_VEL
LIN {X 0,Y 594.365,Z 109.257,A -85,B 0,C 180,E1 -1213.3,E2 -1213.3} C_VEL
LIN {X 0,Y 594.361,Z 109.259,A -85,B 0,C 180,E1 -1216.161,E2 -1216.161} C_VEL
LIN {X 0,Y 594.378,Z 109.254,A -85,B 0,C 180,E1 -1218.536,E2 -1218.536} C_VEL
LIN {X 0,Y 594.381,Z 109.259,A -85,B 0,C 180,E1 -1221.296,E2 -1221.296} C_VEL
LIN {X 0,Y 594.395,Z 109.256,A -85,B 0,C 180,E1 -1223.759,E2 -1223.759} C_VEL
LIN {X 0,Y 594.376,Z 109.254,A -85,B 0,C 180,E1 -1226.239,E2 -1226.239} C_VEL
LIN {X 0,Y 594.369,Z 109.256,A -85,B 0,C 180,E1 -1228.65,E2 -1228.65} C_VEL
LIN {X 0,Y 594.384,Z 109.261,A -85,B 0,C 180,E1 -1231.042,E2 -1231.042} C_VEL
LIN {X 0,Y 594.383,Z 109.259,A -85,B 0,C 180,E1 -1233.3,E2 -1233.3} C_VEL
LIN {X 0,Y 594.377,Z 109.255,A -85,B 0,C 180,E1 -1236.295,E2 -1236.295} C_VEL
LIN {X 0,Y 594.405,Z 109.254,A -85,B 0,C 180,E1 -1239.225,E2 -1239.225} C_VEL
LIN {X 0,Y 594.348,Z 109.259,A -85,B 0,C 180,E1 -1242.095,E2 -1242.095} C_VEL
LIN {X 0,Y 594.365,Z 109.258,A -85,B 0,C 180,E1 -1244.219,E2 -1244.219} C_VEL
LIN {X 0,Y 594.379,Z 109.259,A -85,B 0,C 180,E1 -1246.321,E2 -1246.321} C_VEL
LIN {X 0,Y 594.378,Z 109.255,A -85,B 0,C 180,E1 -1249.095,E2 -1249.095} C_VEL
LIN {X 0,Y 594.413,Z 109.252,A -85,B 0,C 180,E1 -1251.843,E2 -1251.843} C_VEL
LIN {X 0,Y 594.39,Z 109.257,A -85,B 0,C 180,E1 -1254.572,E2 -1254.572} C_VEL
LIN {X 0,Y 594.404,Z 109.25,A -85,B 0,C 180,E1 -1257.289,E2 -1257.289} C_VEL
LIN {X 0,Y 594.415,Z 109.258,A -85,B 0,C 180,E1 -1260,E2 -1260} C_VEL
LIN {X 0,Y 594.405,Z 109.251,A -85,B 0,C 180,E1 -1262.711,E2 -1262.711} C_VEL
LIN {X 0,Y 594.388,Z 109.256,A -85,B 0,C 180,E1 -1265.428,E2 -1265.428} C_VEL
LIN {X 0,Y 594.415,Z 109.253,A -85,B 0,C 180,E1 -1268.157,E2 -1268.157} C_VEL
LIN {X 0,Y 594.392,Z 109.254,A -85,B 0,C 180,E1 -1271.074,E2 -1271.074} C_VEL
LIN {X 0,Y 594.377,Z 109.262,A -85,B 0,C 180,E1 -1273.679,E2 -1273.679} C_VEL
LIN {X 0,Y 594.361,Z 109.258,A -85,B 0,C 180,E1 -1275.323,E2 -1275.323} C_VEL
LIN {X 0,Y 593.685,Z 109.344,A -85,B 0,C 180,E1 -1275.889,E2 -1275.889} C_VEL
LIN {X 0,Y 590.819,Z 109.7,A -85,B 0,C 180,E1 -1276.807,E2 -1276.807} C_VEL
LIN {X 0,Y 588.409,Z 110.005,A -85,B 0,C 180,E1 -1277.545,E2 -1277.545} C_VEL
LIN {X 0,Y 587.387,Z 110.126,A -85,B 0,C 180,E1 -1278.115,E2 -1278.115} C_VEL
LIN {X 0,Y 587.31,Z 110.134,A -85,B 0,C 180,E1 -1278.308,E2 -1278.308} C_VEL
LIN {X 0,Y 587.333,Z 110.137,A -85,B 0,C 180,E1 -1281.038,E2 -1281.038} C_VEL
LIN {X 0,Y 587.316,Z 110.142,A -85,B 0,C 180,E1 -1283.259,E2 -1283.259} C_VEL
LIN {X 0,Y 587.332,Z 110.135,A -85,B 0,C 180,E1 -1285.517,E2 -1285.517} C_VEL
LIN {X 0,Y 587.348,Z 110.13,A -85,B 0,C 180,E1 -1287.818,E2 -1287.818} C_VEL
LIN {X 0,Y 587.339,Z 110.134,A -85,B 0,C 180,E1 -1290.51,E2 -1290.51} C_VEL
LIN {X 0,Y 587.334,Z 110.133,A -85,B 0,C 180,E1 -1293.397,E2 -1293.397} C_VEL
LIN {X 0,Y 587.321,Z 110.133,A -85,B 0,C 180,E1 -1295.898,E2 -1295.898} C_VEL
LIN {X 0,Y 587.329,Z 110.139,A -85,B 0,C 180,E1 -1298.48,E2 -1298.48} C_VEL
LIN {X 0,Y 587.336,Z 110.132,A -85,B 0,C 180,E1 -1301.157,E2 -1301.157} C_VEL
LIN {X 0,Y 587.313,Z 110.139,A -85,B 0,C 180,E1 -1304.112,E2 -1304.112} C_VEL
LIN {X 0,Y 587.314,Z 110.135,A -85,B 0,C 180,E1 -1306.993,E2 -1306.993} C_VEL
LIN {X 0,Y 587.313,Z 110.137,A -85,B 0,C 180,E1 -1309.745,E2 -1309.745} C_VEL
LIN {X 0,Y 587.345,Z 110.135,A -85,B 0,C 180,E1 -1312.392,E2 -1312.392} C_VEL
LIN {X 0,Y 587.336,Z 110.131,A -85,B 0,C 180,E1 -1314.945,E2 -1314.945} C_VEL
LIN {X 0,Y 587.339,Z 110.133,A -85,B 0,C 180,E1 -1317.421,E2 -1317.421} C_VEL
LIN {X 0,Y 587.335,Z 110.141,A -85,B 0,C 180,E1 -1319.83,E2 -1319.83} C_VEL
LIN {X 0,Y 587.354,Z 110.13,A -85,B 0,C 180,E1 -1322.307,E2 -1322.307} C_VEL
LIN {X 0,Y 587.352,Z 110.133,A -85,B 0,C 180,E1 -1325.241,E2 -1325.241} C_VEL
LIN {X 0,Y 587.323,Z 110.134,A -85,B 0,C 180,E1 -1328.226,E2 -1328.226} C_VEL
LIN {X 0,Y 587.38,Z 110.292,A -85,B 0,C 180,E1 -1331.243,E2 -1331.243} C_VEL
LIN {X 0,Y 587.389,Z 122.459,A -85,B 0,C 180,E1 -1333.67,E2 -1333.67} C_VEL
LIN {X 0,Y 587.342,Z 136.947,A -85,B 0,C 180,E1 -1336.507,E2 -1336.507} C_VEL
LIN {X 0,Y 587.236,Z 151.483,A -85,B 0,C 180,E1 -1339.314,E2 -1339.314} C_VEL
LIN {X 0,Y 587.288,Z 152.638,A -85,B 0,C 180,E1 -1339.444,E2 -1339.444} C_VEL
LIN {X 0,Y 587.584,Z 156.926,A -85,B 0,C 180,E1 -1339.514,E2 -1339.514} C_VEL
LIN {X 0,Y 587.545,Z 228.348,A -85,B 0,C 180,E1 -1340.403,E2 -1340.403} C_VEL
LIN {X 0,Y 587.496,Z 238.852,A -85,B 0,C 180,E1 -1340.641,E2 -1340.641} C_VEL
LIN {X 0,Y 587.454,Z 250.553,A -85,B 0,C 180,E1 -1341.053,E2 -1341.053} C_VEL
LIN {X 0,Y 587.395,Z 260.953,A -85,B 0,C 180,E1 -1341.572,E2 -1341.572} C_VEL
LIN {X 0,Y 587.334,Z 269.137,A -85,B 0,C 180,E1 -1342.09,E2 -1342.09} C_VEL
LIN {X 0,Y 587.291,Z 276.892,A -85,B 0,C 180,E1 -1342.695,E2 -1342.695} C_VEL
LIN {X 0,Y 587.286,Z 284.719,A -85,B 0,C 180,E1 -1343.443,E2 -1343.443} C_VEL
LIN {X 0,Y 587.238,Z 292.123,A -85,B 0,C 180,E1 -1344.334,E2 -1344.334} C_VEL
LIN {X 0,Y 587.173,Z 297.736,A -85,B 0,C 180,E1 -1345.194,E2 -1345.194} C_VEL
LIN {X 0,Y 587.211,Z 302.949,A -85,B 0,C 180,E1 -1346.226,E2 -1346.226} C_VEL
LIN {X 0,Y 587.157,Z 305.639,A -85,B 0,C 180,E1 -1346.912,E2 -1346.912} C_VEL
LIN {X 0,Y 587.141,Z 308.577,A -85,B 0,C 180,E1 -1347.942,E2 -1347.942} C_VEL
LIN {X 0,Y 587.144,Z 309.873,A -85,B 0,C 180,E1 -1348.628,E2 -1348.628} C_VEL
LIN {X 0,Y 587.136,Z 310.69,A -85,B 0,C 180,E1 -1349.314,E2 -1349.314} C_VEL
LIN {X 0,Y 587.135,Z 310.996,A -85,B 0,C 180,E1 -1350,E2 -1350} C_VEL
LIN {X 0,Y 587.137,Z 310.732,A -85,B 0,C 180,E1 -1350.686,E2 -1350.686} C_VEL
LIN {X 0,Y 587.146,Z 309.999,A -85,B 0,C 180,E1 -1351.372,E2 -1351.372} C_VEL
LIN {X 0,Y 587.141,Z 308.788,A -85,B 0,C 180,E1 -1352.058,E2 -1352.058} C_VEL
LIN {X 0,Y 587.156,Z 305.941,A -85,B 0,C 180,E1 -1353.087,E2 -1353.087} C_VEL
LIN {X 0,Y 587.211,Z 303.348,A -85,B 0,C 180,E1 -1353.774,E2 -1353.774} C_VEL
LIN {X 0,Y 587.17,Z 298.238,A -85,B 0,C 180,E1 -1354.806,E2 -1354.806} C_VEL
LIN {X 0,Y 587.239,Z 292.74,A -85,B 0,C 180,E1 -1355.666,E2 -1355.666} C_VEL
LIN {X 0,Y 587.268,Z 284.751,A -85,B 0,C 180,E1 -1356.644,E2 -1356.644} C_VEL
LIN {X 0,Y 587.297,Z 276.938,A -85,B 0,C 180,E1 -1357.391,E2 -1357.391} C_VEL
LIN {X 0,Y 587.342,Z 269.191,A -85,B 0,C 180,E1 -1357.996,E2 -1357.996} C_VEL
LIN {X 0,Y 587.395,Z 261.018,A -85,B 0,C 180,E1 -1358.515,E2 -1358.515} C_VEL
LIN {X 0,Y 587.458,Z 250.63,A -85,B 0,C 180,E1 -1359.034,E2 -1359.034} C_VEL
LIN {X 0,Y 587.511,Z 238.986,A -85,B 0,C 180,E1 -1359.445,E2 -1359.445} C_VEL
LIN {X 0,Y 587.548,Z 228.553,A -85,B 0,C 180,E1 -1359.684,E2 -1359.684} C_VEL
LIN {X 0,Y 587.567,Z 173.161,A -85,B 0,C 180,E1 -1360.379,E2 -1360.379} C_VEL
LIN {X 0,Y 587.445,Z 153.761,A -85,B 0,C 180,E1 -1360.617,E2 -1360.617} C_VEL
LIN {X 0,Y 587.246,Z 152.084,A -85,B 0,C 180,E1 -1360.685,E2 -1360.685} C_VEL
LIN {X 0,Y 587.276,Z 139.223,A -85,B 0,C 180,E1 -1363.142,E2 -1363.142} C_VEL
LIN {X 0,Y 587.338,Z 126.54,A -85,B 0,C 180,E1 -1365.618,E2 -1365.618} C_VEL
LIN {X 0,Y 587.467,Z 112.045,A -85,B 0,C 180,E1 -1368.483,E2 -1368.483} C_VEL
LIN {X 0,Y 587.382,Z 110.183,A -85,B 0,C 180,E1 -1368.899,E2 -1368.899} C_VEL
LIN {X 0,Y 587.319,Z 110.134,A -85,B 0,C 180,E1 -1371.774,E2 -1371.774} C_VEL
LIN {X 0,Y 587.35,Z 110.134,A -85,B 0,C 180,E1 -1374.758,E2 -1374.758} C_VEL
LIN {X 0,Y 587.348,Z 110.132,A -85,B 0,C 180,E1 -1377.817,E2 -1377.817} C_VEL
LIN {X 0,Y 587.337,Z 110.136,A -85,B 0,C 180,E1 -1380.51,E2 -1380.51} C_VEL
LIN {X 0,Y 587.328,Z 110.133,A -85,B 0,C 180,E1 -1383.397,E2 -1383.397} C_VEL
LIN {X 0,Y 587.3,Z 110.143,A -85,B 0,C 180,E1 -1385.899,E2 -1385.899} C_VEL
LIN {X 0,Y 587.329,Z 110.134,A -85,B 0,C 180,E1 -1388.479,E2 -1388.479} C_VEL
LIN {X 0,Y 587.334,Z 110.132,A -85,B 0,C 180,E1 -1391.157,E2 -1391.157} C_VEL
LIN {X 0,Y 587.311,Z 110.138,A -85,B 0,C 180,E1 -1394.112,E2 -1394.112} C_VEL
LIN {X 0,Y 587.313,Z 110.135,A -85,B 0,C 180,E1 -1396.993,E2 -1396.993} C_VEL
LIN {X 0,Y 587.312,Z 110.14,A -85,B 0,C 180,E1 -1399.745,E2 -1399.745} C_VEL
LIN {X 0,Y 587.343,Z 110.13,A -85,B 0,C 180,E1 -1402.392,E2 -1402.392} C_VEL
LIN {X 0,Y 587.329,Z 110.136,A -85,B 0,C 180,E1 -1404.944,E2 -1404.944} C_VEL
LIN {X 0,Y 587.336,Z 110.137,A -85,B 0,C 180,E1 -1407.421,E2 -1407.421} C_VEL
LIN {X 0,Y 587.333,Z 110.132,A -85,B 0,C 180,E1 -1409.83,E2 -1409.83} C_VEL
LIN {X 0,Y 587.35,Z 110.13,A -85,B 0,C 180,E1 -1412.307,E2 -1412.307} C_VEL
LIN {X 0,Y 587.35,Z 110.134,A -85,B 0,C 180,E1 -1415.241,E2 -1415.241} C_VEL
LIN {X 0,Y 587.321,Z 110.134,A -85,B 0,C 180,E1 -1418.226,E2 -1418.226} C_VEL
LIN {X 0,Y 587.349,Z 110.132,A -85,B 0,C 180,E1 -1421.151,E2 -1421.151} C_VEL
LIN {X 0,Y 587.323,Z 110.134,A -85,B 0,C 180,E1 -1424.025,E2 -1424.025} C_VEL
LIN {X 0,Y 587.357,Z 110.133,A -85,B 0,C 180,E1 -1426.154,E2 -1426.154} C_VEL
LIN {X 0,Y 587.342,Z 110.132,A -85,B 0,C 180,E1 -1428.962,E2 -1428.962} C_VEL
LIN {X 0,Y 587.365,Z 110.129,A -85,B 0,C 180,E1 -1431.745,E2 -1431.745} C_VEL
LIN {X 0,Y 587.356,Z 110.133,A -85,B 0,C 180,E1 -1434.507,E2 -1434.507} C_VEL
LIN {X 0,Y 587.371,Z 110.127,A -85,B 0,C 180,E1 -1437.257,E2 -1437.257} C_VEL
LIN {X 0,Y 587.383,Z 110.135,A -85,B 0,C 180,E1 -1440,E2 -1440} C_VEL
LIN {X 0,Y 587.37,Z 110.127,A -85,B 0,C 180,E1 -1442.743,E2 -1442.743} C_VEL
LIN {X 0,Y 587.355,Z 110.134,A -85,B 0,C 180,E1 -1445.493,E2 -1445.493} C_VEL
LIN {X 0,Y 587.365,Z 110.129,A -85,B 0,C 180,E1 -1448.255,E2 -1448.255} C_VEL
LIN {X 0,Y 587.347,Z 110.133,A -85,B 0,C 180,E1 -1451.134,E2 -1451.134} C_VEL
LIN {X 0,Y 587.363,Z 110.128,A -85,B 0,C 180,E1 -1454.26,E2 -1454.26} C_VEL
LIN {X 0,Y 587.35,Z 110.137,A -85,B 0,C 180,E1 -1457.406,E2 -1457.406} C_VEL
LIN {X 0,Y 587.329,Z 110.132,A -85,B 0,C 180,E1 -1460.305,E2 -1460.305} C_VEL
LIN {X 0,Y 587.313,Z 110.141,A -85,B 0,C 180,E1 -1463.259,E2 -1463.259} C_VEL
LIN {X 0,Y 587.329,Z 110.134,A -85,B 0,C 180,E1 -1465.517,E2 -1465.517} C_VEL
LIN {X 0,Y 587.346,Z 110.13,A -85,B 0,C 180,E1 -1467.818,E2 -1467.818} C_VEL
LIN {X 0,Y 587.335,Z 110.136,A -85,B 0,C 180,E1 -1470.51,E2 -1470.51} C_VEL
LIN {X 0,Y 587.331,Z 110.132,A -85,B 0,C 180,E1 -1473.397,E2 -1473.397} C_VEL
LIN {X 0,Y 587.317,Z 110.134,A -85,B 0,C 180,E1 -1475.898,E2 -1475.898} C_VEL
LIN {X 0,Y 587.327,Z 110.142,A -85,B 0,C 180,E1 -1478.48,E2 -1478.48} C_VEL
LIN {X 0,Y 587.333,Z 110.132,A -85,B 0,C 180,E1 -1481.157,E2 -1481.157} C_VEL
LIN {X 0,Y 587.325,Z 110.139,A -85,B 0,C 180,E1 -1484.114,E2 -1484.114} C_VEL
LIN {X 0,Y 587.311,Z 110.134,A -85,B 0,C 180,E1 -1486.994,E2 -1486.994} C_VEL
LIN {X 0,Y 587.312,Z 110.139,A -85,B 0,C 180,E1 -1489.746,E2 -1489.746} C_VEL
LIN {X 0,Y 587.342,Z 110.134,A -85,B 0,C 180,E1 -1492.392,E2 -1492.392} C_VEL
LIN {X 0,Y 587.333,Z 110.131,A -85,B 0,C 180,E1 -1494.945,E2 -1494.945} C_VEL
LIN {X 0,Y 587.338,Z 110.135,A -85,B 0,C 180,E1 -1497.421,E2 -1497.421} C_VEL
LIN {X 0,Y 587.331,Z 110.139,A -85,B 0,C 180,E1 -1499.83,E2 -1499.83} C_VEL
LIN {X 0,Y 587.351,Z 110.13,A -85,B 0,C 180,E1 -1502.307,E2 -1502.307} C_VEL
LIN {X 0,Y 587.349,Z 110.136,A -85,B 0,C 180,E1 -1505.242,E2 -1505.242} C_VEL
LIN {X 0,Y 587.318,Z 110.138,A -85,B 0,C 180,E1 -1508.226,E2 -1508.226} C_VEL
LIN {X 0,Y 587.38,Z 110.287,A -85,B 0,C 180,E1 -1509.003,E2 -1509.003} C_VEL
LIN {X 0,Y 587.6,Z 117.349,A -85,B 0,C 180,E1 -1510.252,E2 -1510.252} C_VEL
LIN {X 0,Y 587.428,Z 134.241,A -85,B 0,C 180,E1 -1513.161,E2 -1513.161} C_VEL
LIN {X 0,Y 587.356,Z 150.115,A -85,B 0,C 180,E1 -1515.857,E2 -1515.857} C_VEL
LIN {X 0,Y 587.278,Z 166.527,A -85,B 0,C 180,E1 -1518.612,E2 -1518.612} C_VEL
LIN {X 0,Y 587.279,Z 171.144,A -85,B 0,C 180,E1 -1519.357,E2 -1519.357} C_VEL
LIN {X 0,Y 587.555,Z 173.497,A -85,B 0,C 180,E1 -1519.427,E2 -1519.427} C_VEL
LIN {X 0,Y 587.56,Z 247.151,A -85,B 0,C 180,E1 -1520.338,E2 -1520.338} C_VEL
LIN {X 0,Y 587.497,Z 256.421,A -85,B 0,C 180,E1 -1520.533,E2 -1520.533} C_VEL
LIN {X 0,Y 587.445,Z 264.897,A -85,B 0,C 180,E1 -1520.792,E2 -1520.792} C_VEL
LIN {X 0,Y 587.418,Z 273.405,A -85,B 0,C 180,E1 -1521.139,E2 -1521.139} C_VEL
LIN {X 0,Y 587.394,Z 281.734,A -85,B 0,C 180,E1 -1521.572,E2 -1521.572} C_VEL
LIN {X 0,Y 587.333,Z 289.77,A -85,B 0,C 180,E1 -1522.091,E2 -1522.091} C_VEL
LIN {X 0,Y 587.291,Z 297.419,A -85,B 0,C 180,E1 -1522.695,E2 -1522.695} C_VEL
LIN {X 0,Y 587.281,Z 305.809,A -85,B 0,C 180,E1 -1523.512,E2 -1523.512} C_VEL
LIN {X 0,Y 587.239,Z 312.434,A -85,B 0,C 180,E1 -1524.334,E2 -1524.334} C_VEL
LIN {X 0,Y 587.17,Z 317.988,A -85,B 0,C 180,E1 -1525.194,E2 -1525.194} C_VEL
LIN {X 0,Y 587.21,Z 323.148,A -85,B 0,C 180,E1 -1526.226,E2 -1526.226} C_VEL
LIN {X 0,Y 587.155,Z 325.789,A -85,B 0,C 180,E1 -1526.913,E2 -1526.913} C_VEL
LIN {X 0,Y 587.14,Z 328.681,A -85,B 0,C 180,E1 -1527.942,E2 -1527.942} C_VEL
LIN {X 0,Y 587.145,Z 329.937,A -85,B 0,C 180,E1 -1528.628,E2 -1528.628} C_VEL
LIN {X 0,Y 587.136,Z 330.711,A -85,B 0,C 180,E1 -1529.314,E2 -1529.314} C_VEL
LIN {X 0,Y 587.134,Z 331,A -85,B 0,C 180,E1 -1530,E2 -1530} C_VEL
LIN {X 0,Y 587.136,Z 330.711,A -85,B 0,C 180,E1 -1530.686,E2 -1530.686} C_VEL
LIN {X 0,Y 587.145,Z 329.936,A -85,B 0,C 180,E1 -1531.372,E2 -1531.372} C_VEL
LIN {X 0,Y 587.14,Z 328.68,A -85,B 0,C 180,E1 -1532.058,E2 -1532.058} C_VEL
LIN {X 0,Y 587.155,Z 325.788,A -85,B 0,C 180,E1 -1533.088,E2 -1533.088} C_VEL
LIN {X 0,Y 587.21,Z 323.147,A -85,B 0,C 180,E1 -1533.774,E2 -1533.774} C_VEL
LIN {X 0,Y 587.17,Z 317.985,A -85,B 0,C 180,E1 -1534.806,E2 -1534.806} C_VEL
LIN {X 0,Y 587.253,Z 311.186,A -85,B 0,C 180,E1 -1535.839,E2 -1535.839} C_VEL
LIN {X 0,Y 587.269,Z 304.285,A -85,B 0,C 180,E1 -1536.646,E2 -1536.646} C_VEL
LIN {X 0,Y 587.296,Z 296.405,A -85,B 0,C 180,E1 -1537.391,E2 -1537.391} C_VEL
LIN {X 0,Y 587.342,Z 288.545,A -85,B 0,C 180,E1 -1537.996,E2 -1537.996} C_VEL
LIN {X 0,Y 587.435,Z 278.73,A -85,B 0,C 180,E1 -1538.601,E2 -1538.601} C_VEL
LIN {X 0,Y 587.463,Z 267.297,A -85,B 0,C 180,E1 -1539.121,E2 -1539.121} C_VEL
LIN {X 0,Y 587.505,Z 257.24,A -85,B 0,C 180,E1 -1539.446,E2 -1539.446} C_VEL
LIN {X 0,Y 587.541,Z 248.434,A -85,B 0,C 180,E1 -1539.641,E2 -1539.641} C_VEL
LIN {X 0,Y 587.579,Z 175.311,A -85,B 0,C 180,E1 -1540.551,E2 -1540.551} C_VEL
LIN {X 0,Y 587.29,Z 171.455,A -85,B 0,C 180,E1 -1540.62,E2 -1540.62} C_VEL
LIN {X 0,Y 587.281,Z 168.251,A -85,B 0,C 180,E1 -1541.1,E2 -1541.1} C_VEL
LIN {X 0,Y 587.39,Z 151.875,A -85,B 0,C 180,E1 -1543.845,E2 -1543.845} C_VEL
LIN {X 0,Y 587.444,Z 135.134,A -85,B 0,C 180,E1 -1546.686,E2 -1546.686} C_VEL
LIN {X 0,Y 587.573,Z 118.393,A -85,B 0,C 180,E1 -1549.567,E2 -1549.567} C_VEL
LIN {X 0,Y 587.404,Z 110.453,A -85,B 0,C 180,E1 -1550.958,E2 -1550.958} C_VEL
LIN {X 0,Y 587.361,Z 110.187,A -85,B 0,C 180,E1 -1551.045,E2 -1551.045} C_VEL
LIN {X 0,Y 587.315,Z 110.129,A -85,B 0,C 180,E1 -1554.008,E2 -1554.008} C_VEL
LIN {X 0,Y 587.337,Z 110.138,A -85,B 0,C 180,E1 -1556.279,E2 -1556.279} C_VEL
LIN {X 0,Y 587.35,Z 110.13,A -85,B 0,C 180,E1 -1559.133,E2 -1559.133} C_VEL
LIN {X 0,Y 587.344,Z 110.133,A -85,B 0,C 180,E1 -1561.835,E2 -1561.835} C_VEL
LIN {X 0,Y 587.346,Z 110.137,A -85,B 0,C 180,E1 -1564.347,E2 -1564.347} C_VEL
LIN {X 0,Y 587.344,Z 110.133,A -85,B 0,C 180,E1 -1567.608,E2 -1567.608} C_VEL
LIN {X 0,Y 587.313,Z 110.139,A -85,B 0,C 180,E1 -1570.255,E2 -1570.255} C_VEL
LIN {X 0,Y 587.314,Z 110.134,A -85,B 0,C 180,E1 -1573.118,E2 -1573.118} C_VEL
LIN {X 0,Y 587.313,Z 110.138,A -85,B 0,C 180,E1 -1576.049,E2 -1576.049} C_VEL
LIN {X 0,Y 587.334,Z 110.132,A -85,B 0,C 180,E1 -1578.925,E2 -1578.925} C_VEL
LIN {X 0,Y 587.328,Z 110.142,A -85,B 0,C 180,E1 -1581.521,E2 -1581.521} C_VEL
LIN {X 0,Y 587.319,Z 110.134,A -85,B 0,C 180,E1 -1584.102,E2 -1584.102} C_VEL
LIN {X 0,Y 587.338,Z 110.134,A -85,B 0,C 180,E1 -1586.889,E2 -1586.889} C_VEL
LIN {X 0,Y 587.334,Z 110.133,A -85,B 0,C 180,E1 -1589.83,E2 -1589.83} C_VEL
LIN {X 0,Y 587.352,Z 110.129,A -85,B 0,C 180,E1 -1592.307,E2 -1592.307} C_VEL
LIN {X 0,Y 587.351,Z 110.135,A -85,B 0,C 180,E1 -1595.242,E2 -1595.242} C_VEL
LIN {X 0,Y 587.321,Z 110.134,A -85,B 0,C 180,E1 -1598.226,E2 -1598.226} C_VEL
LIN {X 0,Y 587.349,Z 110.133,A -85,B 0,C 180,E1 -1601.151,E2 -1601.151} C_VEL
LIN {X 0,Y 587.323,Z 110.134,A -85,B 0,C 180,E1 -1604.025,E2 -1604.025} C_VEL
LIN {X 0,Y 587.358,Z 110.131,A -85,B 0,C 180,E1 -1606.154,E2 -1606.154} C_VEL
LIN {X 0,Y 587.344,Z 110.133,A -85,B 0,C 180,E1 -1608.963,E2 -1608.963} C_VEL
LIN {X 0,Y 587.366,Z 110.129,A -85,B 0,C 180,E1 -1611.745,E2 -1611.745} C_VEL
LIN {X 0,Y 587.355,Z 110.135,A -85,B 0,C 180,E1 -1614.507,E2 -1614.507} C_VEL
LIN {X 0,Y 587.371,Z 110.127,A -85,B 0,C 180,E1 -1617.257,E2 -1617.257} C_VEL
LIN {X 0,Y 587.384,Z 110.134,A -85,B 0,C 180,E1 -1620,E2 -1620} C_VEL
LIN {X 0,Y 587.371,Z 110.127,A -85,B 0,C 180,E1 -1622.743,E2 -1622.743} C_VEL
LIN {X 0,Y 587.355,Z 110.133,A -85,B 0,C 180,E1 -1625.493,E2 -1625.493} C_VEL
LIN {X 0,Y 587.367,Z 110.13,A -85,B 0,C 180,E1 -1628.255,E2 -1628.255} C_VEL
LIN {X 0,Y 587.35,Z 110.131,A -85,B 0,C 180,E1 -1631.134,E2 -1631.134} C_VEL
LIN {X 0,Y 587.366,Z 110.128,A -85,B 0,C 180,E1 -1634.26,E2 -1634.26} C_VEL
LIN {X 0,Y 587.351,Z 110.139,A -85,B 0,C 180,E1 -1637.406,E2 -1637.406} C_VEL
LIN {X 0,Y 587.31,Z 110.134,A -85,B 0,C 180,E1 -1638.308,E2 -1638.308} C_VEL
LIN {X 0,Y 586.668,Z 110.217,A -85,B 0,C 180,E1 -1638.88,E2 -1638.88} C_VEL
LIN {X 0,Y 583.844,Z 110.578,A -85,B 0,C 180,E1 -1639.809,E2 -1639.809} C_VEL
LIN {X 0,Y 581.434,Z 110.883,A -85,B 0,C 180,E1 -1640.556,E2 -1640.556} C_VEL
LIN {X 0,Y 580.38,Z 111.01,A -85,B 0,C 180,E1 -1641.132,E2 -1641.132} C_VEL
LIN {X 0,Y 580.285,Z 111.018,A -85,B 0,C 180,E1 -1641.328,E2 -1641.328} C_VEL
LIN {X 0,Y 580.299,Z 111.008,A -85,B 0,C 180,E1 -1644.316,E2 -1644.316} C_VEL
LIN {X 0,Y 580.278,Z 111.013,A -85,B 0,C 180,E1 -1646.623,E2 -1646.623} C_VEL
LIN {X 0,Y 580.303,Z 111.011,A -85,B 0,C 180,E1 -1649.31,E2 -1649.31} C_VEL
LIN {X 0,Y 580.299,Z 111.009,A -85,B 0,C 180,E1 -1652.201,E2 -1652.201} C_VEL
LIN {X 0,Y 580.294,Z 111.017,A -85,B 0,C 180,E1 -1654.696,E2 -1654.696} C_VEL
LIN {X 0,Y 580.3,Z 111.009,A -85,B 0,C 180,E1 -1657.268,E2 -1657.268} C_VEL
LIN {X 0,Y 580.293,Z 111.013,A -85,B 0,C 180,E1 -1660.27,E2 -1660.27} C_VEL
LIN {X 0,Y 580.278,Z 111.016,A -85,B 0,C 180,E1 -1662.706,E2 -1662.706} C_VEL
LIN {X 0,Y 580.256,Z 111.013,A -85,B 0,C 180,E1 -1665.611,E2 -1665.611} C_VEL
LIN {X 0,Y 580.281,Z 111.019,A -85,B 0,C 180,E1 -1668.231,E2 -1668.231} C_VEL
LIN {X 0,Y 580.279,Z 111.01,A -85,B 0,C 180,E1 -1670.965,E2 -1670.965} C_VEL
LIN {X 0,Y 580.274,Z 111.014,A -85,B 0,C 180,E1 -1673.597,E2 -1673.597} C_VEL
LIN {X 0,Y 580.305,Z 111.014,A -85,B 0,C 180,E1 -1676.144,E2 -1676.144} C_VEL
LIN {X 0,Y 580.277,Z 111.011,A -85,B 0,C 180,E1 -1678.614,E2 -1678.614} C_VEL
LIN {X 0,Y 580.294,Z 111.009,A -85,B 0,C 180,E1 -1681.024,E2 -1681.024} C_VEL
LIN {X 0,Y 580.292,Z 111.018,A -85,B 0,C 180,E1 -1683.666,E2 -1683.666} C_VEL
LIN {X 0,Y 580.299,Z 111.017,A -85,B 0,C 180,E1 -1685.684,E2 -1685.684} C_VEL
LIN {X 0,Y 580.288,Z 111.01,A -85,B 0,C 180,E1 -1688.695,E2 -1688.695} C_VEL
LIN {X 0,Y 580.346,Z 111.147,A -85,B 0,C 180,E1 -1691.19,E2 -1691.19} C_VEL
LIN {X 0,Y 580.362,Z 122.461,A -85,B 0,C 180,E1 -1693.466,E2 -1693.466} C_VEL
LIN {X 0,Y 580.293,Z 136.95,A -85,B 0,C 180,E1 -1696.339,E2 -1696.339} C_VEL
LIN {X 0,Y 580.176,Z 151.734,A -85,B 0,C 180,E1 -1699.224,E2 -1699.224} C_VEL
LIN {X 0,Y 580.233,Z 152.821,A -85,B 0,C 180,E1 -1699.321,E2 -1699.321} C_VEL
LIN {X 0,Y 580.622,Z 156.875,A -85,B 0,C 180,E1 -1699.386,E2 -1699.386} C_VEL
LIN {X 0,Y 580.57,Z 228.381,A -85,B 0,C 180,E1 -1700.287,E2 -1700.287} C_VEL
LIN {X 0,Y 580.503,Z 238.877,A -85,B 0,C 180,E1 -1700.527,E2 -1700.527} C_VEL
LIN {X 0,Y 580.436,Z 250.561,A -85,B 0,C 180,E1 -1700.944,E2 -1700.944} C_VEL
LIN {X 0,Y 580.363,Z 260.959,A -85,B 0,C 180,E1 -1701.469,E2 -1701.469} C_VEL
LIN {X 0,Y 580.285,Z 269.141,A -85,B 0,C 180,E1 -1701.994,E2 -1701.994} C_VEL
LIN {X 0,Y 580.241,Z 276.901,A -85,B 0,C 180,E1 -1702.606,E2 -1702.606} C_VEL
LIN {X 0,Y 580.21,Z 284.518,A -85,B 0,C 180,E1 -1703.342,E2 -1703.342} C_VEL
LIN {X 0,Y 580.173,Z 292.128,A -85,B 0,C 180,E1 -1704.264,E2 -1704.264} C_VEL
LIN {X 0,Y 580.088,Z 297.739,A -85,B 0,C 180,E1 -1705.135,E2 -1705.135} C_VEL
LIN {X 0,Y 580.138,Z 302.953,A -85,B 0,C 180,E1 -1706.179,E2 -1706.179} C_VEL
LIN {X 0,Y 580.072,Z 305.64,A -85,B 0,C 180,E1 -1706.874,E2 -1706.874} C_VEL
LIN {X 0,Y 580.04,Z 308.58,A -85,B 0,C 180,E1 -1707.917,E2 -1707.917} C_VEL
LIN {X 0,Y 580.044,Z 309.873,A -85,B 0,C 180,E1 -1708.611,E2 -1708.611} C_VEL
LIN {X 0,Y 580.036,Z 310.69,A -85,B 0,C 180,E1 -1709.306,E2 -1709.306} C_VEL
LIN {X 0,Y 580.036,Z 310.996,A -85,B 0,C 180,E1 -1710,E2 -1710} C_VEL
LIN {X 0,Y 580.037,Z 310.731,A -85,B 0,C 180,E1 -1710.694,E2 -1710.694} C_VEL
LIN {X 0,Y 580.045,Z 309.998,A -85,B 0,C 180,E1 -1711.388,E2 -1711.388} C_VEL
LIN {X 0,Y 580.04,Z 308.788,A -85,B 0,C 180,E1 -1712.083,E2 -1712.083} C_VEL
LIN {X 0,Y 580.071,Z 305.94,A -85,B 0,C 180,E1 -1713.125,E2 -1713.125} C_VEL
LIN {X 0,Y 580.123,Z 303.346,A -85,B 0,C 180,E1 -1713.82,E2 -1713.82} C_VEL
LIN {X 0,Y 580.075,Z 298.236,A -85,B 0,C 180,E1 -1714.865,E2 -1714.865} C_VEL
LIN {X 0,Y 580.174,Z 292.737,A -85,B 0,C 180,E1 -1715.735,E2 -1715.735} C_VEL
LIN {X 0,Y 580.195,Z 285.509,A -85,B 0,C 180,E1 -1716.645,E2 -1716.645} C_VEL
LIN {X 0,Y 580.255,Z 276.934,A -85,B 0,C 180,E1 -1717.481,E2 -1717.481} C_VEL
LIN {X 0,Y 580.308,Z 269.18,A -85,B 0,C 180,E1 -1718.093,E2 -1718.093} C_VEL
LIN {X 0,Y 580.36,Z 261.004,A -85,B 0,C 180,E1 -1718.618,E2 -1718.618} C_VEL
LIN {X 0,Y 580.438,Z 250.615,A -85,B 0,C 180,E1 -1719.144,E2 -1719.144} C_VEL
LIN {X 0,Y 580.518,Z 238.969,A -85,B 0,C 180,E1 -1719.56,E2 -1719.56} C_VEL
LIN {X 0,Y 580.573,Z 228.522,A -85,B 0,C 180,E1 -1719.801,E2 -1719.801} C_VEL
LIN {X 0,Y 580.618,Z 168.91,A -85,B 0,C 180,E1 -1720.556,E2 -1720.556} C_VEL
LIN {X 0,Y 580.392,Z 154.043,A -85,B 0,C 180,E1 -1720.743,E2 -1720.743} C_VEL
LIN {X 0,Y 580.214,Z 152.096,A -85,B 0,C 180,E1 -1720.815,E2 -1720.815} C_VEL
LIN {X 0,Y 580.291,Z 137.408,A -85,B 0,C 180,E1 -1723.66,E2 -1723.66} C_VEL
LIN {X 0,Y 580.339,Z 122.914,A -85,B 0,C 180,E1 -1726.534,E2 -1726.534} C_VEL
LIN {X 0,Y 580.326,Z 111.091,A -85,B 0,C 180,E1 -1728.925,E2 -1728.925} C_VEL
LIN {X 0,Y 580.27,Z 111.015,A -85,B 0,C 180,E1 -1732.052,E2 -1732.052} C_VEL
LIN {X 0,Y 580.304,Z 111.008,A -85,B 0,C 180,E1 -1735.08,E2 -1735.08} C_VEL
LIN {X 0,Y 580.3,Z 111.015,A -85,B 0,C 180,E1 -1738.185,E2 -1738.185} C_VEL
LIN {X 0,Y 580.284,Z 111.012,A -85,B 0,C 180,E1 -1740.694,E2 -1740.694} C_VEL
LIN {X 0,Y 580.283,Z 111.01,A -85,B 0,C 180,E1 -1743.313,E2 -1743.313} C_VEL
LIN {X 0,Y 580.264,Z 111.017,A -85,B 0,C 180,E1 -1745.759,E2 -1745.759} C_VEL
LIN {X 0,Y 580.288,Z 111.016,A -85,B 0,C 180,E1 -1748.146,E2 -1748.146} C_VEL
LIN {X 0,Y 580.297,Z 111.008,A -85,B 0,C 180,E1 -1750.843,E2 -1750.843} C_VEL
LIN {X 0,Y 580.272,Z 111.019,A -85,B 0,C 180,E1 -1753.658,E2 -1753.658} C_VEL
LIN {X 0,Y 580.276,Z 111.01,A -85,B 0,C 180,E1 -1756.609,E2 -1756.609} C_VEL
LIN {X 0,Y 580.296,Z 111.012,A -85,B 0,C 180,E1 -1759.156,E2 -1759.156} C_VEL
LIN {X 0,Y 580.289,Z 111.011,A -85,B 0,C 180,E1 -1761.927,E2 -1761.927} C_VEL
LIN {X 0,Y 580.287,Z 111.009,A -85,B 0,C 180,E1 -1764.455,E2 -1764.455} C_VEL
LIN {X 0,Y 580.289,Z 111.014,A -85,B 0,C 180,E1 -1766.975,E2 -1766.975} C_VEL
LIN {X 0,Y 580.296,Z 111.013,A -85,B 0,C 180,E1 -1769.425,E2 -1769.425} C_VEL
LIN {X 0,Y 580.297,Z 111.008,A -85,B 0,C 180,E1 -1772.141,E2 -1772.141} C_VEL
LIN {X 0,Y 580.321,Z 111.009,A -85,B 0,C 180,E1 -1775.269,E2 -1775.269} C_VEL
LIN {X 0,Y 580.272,Z 111.011,A -85,B 0,C 180,E1 -1777.947,E2 -1777.947} C_VEL
LIN {X 0,Y 580.318,Z 111.011,A -85,B 0,C 180,E1 -1780.914,E2 -1780.914} C_VEL
LIN {X 0,Y 580.278,Z 111.011,A -85,B 0,C 180,E1 -1783.825,E2 -1783.825} C_VEL
LIN {X 0,Y 580.324,Z 111.007,A -85,B 0,C 180,E1 -1785.983,E2 -1785.983} C_VEL
LIN {X 0,Y 580.304,Z 111.01,A -85,B 0,C 180,E1 -1788.827,E2 -1788.827} C_VEL
LIN {X 0,Y 580.328,Z 111.005,A -85,B 0,C 180,E1 -1791.644,E2 -1791.644} C_VEL
LIN {X 0,Y 580.322,Z 111.01,A -85,B 0,C 180,E1 -1794.44,E2 -1794.44} C_VEL
LIN {X 0,Y 580.344,Z 111.01,A -85,B 0,C 180,E1 -1797.918,E2 -1797.918} C_VEL
LIN {X 0,Y 580.36,Z 111.001,A -85,B 0,C 180,E1 -1800.694,E2 -1800.694} C_VEL
LIN {X 0,Y 580.279,Z 111.014,A -85,B 0,C 180,E1 -1803.472,E2 -1803.472} C_VEL
LIN {X 0,Y 580.322,Z 111.011,A -85,B 0,C 180,E1 -1805.56,E2 -1805.56} C_VEL
LIN {X 0,Y 580.328,Z 111.005,A -85,B 0,C 180,E1 -1808.356,E2 -1808.356} C_VEL
LIN {X 0,Y 580.299,Z 111.012,A -85,B 0,C 180,E1 -1811.191,E2 -1811.191} C_VEL
LIN {X 0,Y 580.324,Z 111.006,A -85,B 0,C 180,E1 -1814.017,E2 -1814.017} C_VEL
LIN {X 0,Y 580.311,Z 111.01,A -85,B 0,C 180,E1 -1816.914,E2 -1816.914} C_VEL
LIN {X 0,Y 580.304,Z 111.008,A -85,B 0,C 180,E1 -1819.822,E2 -1819.822} C_VEL
LIN {X 0,Y 580.289,Z 111.014,A -85,B 0,C 180,E1 -1822.803,E2 -1822.803} C_VEL
LIN {X 0,Y 580.304,Z 111.016,A -85,B 0,C 180,E1 -1825.08,E2 -1825.08} C_VEL
LIN {X 0,Y 580.298,Z 111.008,A -85,B 0,C 180,E1 -1828.186,E2 -1828.186} C_VEL
LIN {X 0,Y 580.283,Z 111.018,A -85,B 0,C 180,E1 -1830.695,E2 -1830.695} C_VEL
LIN {X 0,Y 580.301,Z 111.009,A -85,B 0,C 180,E1 -1833.316,E2 -1833.316} C_VEL
LIN {X 0,Y 580.275,Z 111.011,A -85,B 0,C 180,E1 -1835.761,E2 -1835.761} C_VEL
LIN {X 0,Y 580.286,Z 111.013,A -85,B 0,C 180,E1 -1838.146,E2 -1838.146} C_VEL
LIN {X 0,Y 580.296,Z 111.011,A -85,B 0,C 180,E1 -1840.844,E2 -1840.844} C_VEL
LIN {X 0,Y 580.277,Z 111.011,A -85,B 0,C 180,E1 -1843.658,E2 -1843.658} C_VEL
LIN {X 0,Y 580.272,Z 111.014,A -85,B 0,C 180,E1 -1846.61,E2 -1846.61} C_VEL
LIN {X 0,Y 580.295,Z 111.008,A -85,B 0,C 180,E1 -1849.157,E2 -1849.157} C_VEL
LIN {X 0,Y 580.288,Z 111.018,A -85,B 0,C 180,E1 -1851.927,E2 -1851.927} C_VEL
LIN {X 0,Y 580.281,Z 111.012,A -85,B 0,C 180,E1 -1854.455,E2 -1854.455} C_VEL
LIN {X 0,Y 580.288,Z 111.009,A -85,B 0,C 180,E1 -1856.975,E2 -1856.975} C_VEL
LIN {X 0,Y 580.294,Z 111.013,A -85,B 0,C 180,E1 -1859.425,E2 -1859.425} C_VEL
LIN {X 0,Y 580.298,Z 111.01,A -85,B 0,C 180,E1 -1862.141,E2 -1862.141} C_VEL
LIN {X 0,Y 580.32,Z 111.012,A -85,B 0,C 180,E1 -1865.27,E2 -1865.27} C_VEL
LIN {X 0,Y 580.269,Z 111.018,A -85,B 0,C 180,E1 -1867.947,E2 -1867.947} C_VEL
LIN {X 0,Y 580.344,Z 111.176,A -85,B 0,C 180,E1 -1868.916,E2 -1868.916} C_VEL
LIN {X 0,Y 580.613,Z 118.306,A -85,B 0,C 180,E1 -1870.189,E2 -1870.189} C_VEL
LIN {X 0,Y 580.469,Z 133.253,A -85,B 0,C 180,E1 -1872.781,E2 -1872.781} C_VEL
LIN {X 0,Y 580.35,Z 149.917,A -85,B 0,C 180,E1 -1875.649,E2 -1875.649} C_VEL
LIN {X 0,Y 580.24,Z 167.571,A -85,B 0,C 180,E1 -1878.649,E2 -1878.649} C_VEL
LIN {X 0,Y 580.229,Z 171.374,A -85,B 0,C 180,E1 -1879.243,E2 -1879.243} C_VEL
LIN {X 0,Y 580.608,Z 175.795,A -85,B 0,C 180,E1 -1879.327,E2 -1879.327} C_VEL
LIN {X 0,Y 580.556,Z 247.151,A -85,B 0,C 180,E1 -1880.221,E2 -1880.221} C_VEL
LIN {X 0,Y 580.518,Z 256.42,A -85,B 0,C 180,E1 -1880.418,E2 -1880.418} C_VEL
LIN {X 0,Y 580.452,Z 264.895,A -85,B 0,C 180,E1 -1880.681,E2 -1880.681} C_VEL
LIN {X 0,Y 580.42,Z 273.401,A -85,B 0,C 180,E1 -1881.031,E2 -1881.031} C_VEL
LIN {X 0,Y 580.362,Z 281.733,A -85,B 0,C 180,E1 -1881.469,E2 -1881.469} C_VEL
LIN {X 0,Y 580.284,Z 289.772,A -85,B 0,C 180,E1 -1881.994,E2 -1881.994} C_VEL
LIN {X 0,Y 580.224,Z 298.433,A -85,B 0,C 180,E1 -1882.693,E2 -1882.693} C_VEL
LIN {X 0,Y 580.218,Z 306.418,A -85,B 0,C 180,E1 -1883.503,E2 -1883.503} C_VEL
LIN {X 0,Y 580.173,Z 312.435,A -85,B 0,C 180,E1 -1884.265,E2 -1884.265} C_VEL
LIN {X 0,Y 580.084,Z 317.989,A -85,B 0,C 180,E1 -1885.135,E2 -1885.135} C_VEL
LIN {X 0,Y 580.137,Z 323.149,A -85,B 0,C 180,E1 -1886.18,E2 -1886.18} C_VEL
LIN {X 0,Y 580.07,Z 325.789,A -85,B 0,C 180,E1 -1886.875,E2 -1886.875} C_VEL
LIN {X 0,Y 580.04,Z 328.682,A -85,B 0,C 180,E1 -1887.917,E2 -1887.917} C_VEL
LIN {X 0,Y 580.045,Z 329.935,A -85,B 0,C 180,E1 -1888.612,E2 -1888.612} C_VEL
LIN {X 0,Y 580.036,Z 330.71,A -85,B 0,C 180,E1 -1889.306,E2 -1889.306} C_VEL
LIN {X 0,Y 580.034,Z 331,A -85,B 0,C 180,E1 -1890,E2 -1890} C_VEL
LIN {X 0,Y 580.036,Z 330.71,A -85,B 0,C 180,E1 -1890.694,E2 -1890.694} C_VEL
LIN {X 0,Y 580.045,Z 329.934,A -85,B 0,C 180,E1 -1891.389,E2 -1891.389} C_VEL
LIN {X 0,Y 580.04,Z 328.681,A -85,B 0,C 180,E1 -1892.083,E2 -1892.083} C_VEL
LIN {X 0,Y 580.07,Z 325.787,A -85,B 0,C 180,E1 -1893.126,E2 -1893.126} C_VEL
LIN {X 0,Y 580.137,Z 323.147,A -85,B 0,C 180,E1 -1893.821,E2 -1893.821} C_VEL
LIN {X 0,Y 580.084,Z 317.985,A -85,B 0,C 180,E1 -1894.865,E2 -1894.865} C_VEL
LIN {X 0,Y 580.193,Z 311.185,A -85,B 0,C 180,E1 -1895.91,E2 -1895.91} C_VEL
LIN {X 0,Y 580.225,Z 303.494,A -85,B 0,C 180,E1 -1896.808,E2 -1896.808} C_VEL
LIN {X 0,Y 580.254,Z 296.404,A -85,B 0,C 180,E1 -1897.481,E2 -1897.481} C_VEL
LIN {X 0,Y 580.301,Z 288.541,A -85,B 0,C 180,E1 -1898.094,E2 -1898.094} C_VEL
LIN {X 0,Y 580.417,Z 278.727,A -85,B 0,C 180,E1 -1898.706,E2 -1898.706} C_VEL
LIN {X 0,Y 580.455,Z 267.299,A -85,B 0,C 180,E1 -1899.232,E2 -1899.232} C_VEL
LIN {X 0,Y 580.516,Z 257.241,A -85,B 0,C 180,E1 -1899.56,E2 -1899.56} C_VEL
LIN {X 0,Y 580.567,Z 248.433,A -85,B 0,C 180,E1 -1899.757,E2 -1899.757} C_VEL
LIN {X 0,Y 580.595,Z 182.02,A -85,B 0,C 180,E1 -1900.596,E2 -1900.596} C_VEL
LIN {X 0,Y 580.485,Z 173.424,A -85,B 0,C 180,E1 -1900.704,E2 -1900.704} C_VEL
LIN {X 0,Y 580.198,Z 171.121,A -85,B 0,C 180,E1 -1900.777,E2 -1900.777} C_VEL
LIN {X 0,Y 580.298,Z 157.106,A -85,B 0,C 180,E1 -1903.125,E2 -1903.125} C_VEL
LIN {X 0,Y 580.41,Z 141.412,A -85,B 0,C 180,E1 -1905.81,E2 -1905.81} C_VEL
LIN {X 0,Y 580.503,Z 125.693,A -85,B 0,C 180,E1 -1908.53,E2 -1908.53} C_VEL
LIN {X 0,Y 580.602,Z 114.076,A -85,B 0,C 180,E1 -1910.551,E2 -1910.551} C_VEL
LIN {X 0,Y 580.316,Z 111.049,A -85,B 0,C 180,E1 -1911.13,E2 -1911.13} C_VEL
LIN {X 0,Y 580.266,Z 111.001,A -85,B 0,C 180,E1 -1913.559,E2 -1913.559} C_VEL
LIN {X 0,Y 580.278,Z 111.012,A -85,B 0,C 180,E1 -1915.85,E2 -1915.85} C_VEL
LIN {X 0,Y 580.301,Z 111.014,A -85,B 0,C 180,E1 -1918.186,E2 -1918.186} C_VEL
LIN {X 0,Y 580.284,Z 111.013,A -85,B 0,C 180,E1 -1920.694,E2 -1920.694} C_VEL
LIN {X 0,Y 580.284,Z 111.009,A -85,B 0,C 180,E1 -1923.313,E2 -1923.313} C_VEL
LIN {X 0,Y 580.247,Z 111.018,A -85,B 0,C 180,E1 -1925.756,E2 -1925.756} C_VEL
LIN {X 0,Y 580.288,Z 111.017,A -85,B 0,C 180,E1 -1928.146,E2 -1928.146} C_VEL
LIN {X 0,Y 580.297,Z 111.008,A -85,B 0,C 180,E1 -1930.844,E2 -1930.844} C_VEL
LIN {X 0,Y 580.273,Z 111.018,A -85,B 0,C 180,E1 -1933.659,E2 -1933.659} C_VEL
LIN {X 0,Y 580.275,Z 111.011,A -85,B 0,C 180,E1 -1936.61,E2 -1936.61} C_VEL
LIN {X 0,Y 580.297,Z 111.011,A -85,B 0,C 180,E1 -1939.157,E2 -1939.157} C_VEL
LIN {X 0,Y 580.29,Z 111.012,A -85,B 0,C 180,E1 -1941.927,E2 -1941.927} C_VEL
LIN {X 0,Y 580.286,Z 111.009,A -85,B 0,C 180,E1 -1944.455,E2 -1944.455} C_VEL
LIN {X 0,Y 580.29,Z 111.013,A -85,B 0,C 180,E1 -1946.975,E2 -1946.975} C_VEL
LIN {X 0,Y 580.296,Z 111.014,A -85,B 0,C 180,E1 -1949.425,E2 -1949.425} C_VEL
LIN {X 0,Y 580.299,Z 111.007,A -85,B 0,C 180,E1 -1952.141,E2 -1952.141} C_VEL
LIN {X 0,Y 580.322,Z 111.01,A -85,B 0,C 180,E1 -1955.27,E2 -1955.27} C_VEL
LIN {X 0,Y 580.272,Z 111.011,A -85,B 0,C 180,E1 -1957.947,E2 -1957.947} C_VEL
LIN {X 0,Y 580.321,Z 111.013,A -85,B 0,C 180,E1 -1960.914,E2 -1960.914} C_VEL
LIN {X 0,Y 580.279,Z 111.01,A -85,B 0,C 180,E1 -1963.826,E2 -1963.826} C_VEL
LIN {X 0,Y 580.326,Z 111.006,A -85,B 0,C 180,E1 -1965.983,E2 -1965.983} C_VEL
LIN {X 0,Y 580.307,Z 111.011,A -85,B 0,C 180,E1 -1968.827,E2 -1968.827} C_VEL
LIN {X 0,Y 580.329,Z 111.004,A -85,B 0,C 180,E1 -1971.644,E2 -1971.644} C_VEL
LIN {X 0,Y 580.321,Z 111.012,A -85,B 0,C 180,E1 -1974.44,E2 -1974.44} C_VEL
LIN {X 0,Y 580.337,Z 111.003,A -85,B 0,C 180,E1 -1977.224,E2 -1977.224} C_VEL
LIN {X 0,Y 580.354,Z 111.009,A -85,B 0,C 180,E1 -1980,E2 -1980} C_VEL
LIN {X 0,Y 580.337,Z 111.003,A -85,B 0,C 180,E1 -1982.777,E2 -1982.777} C_VEL
LIN {X 0,Y 580.322,Z 111.01,A -85,B 0,C 180,E1 -1985.56,E2 -1985.56} C_VEL
LIN {X 0,Y 580.33,Z 111.005,A -85,B 0,C 180,E1 -1988.356,E2 -1988.356} C_VEL
LIN {X 0,Y 580.302,Z 111.01,A -85,B 0,C 180,E1 -1991.191,E2 -1991.191} C_VEL
LIN {X 0,Y 580.325,Z 111.007,A -85,B 0,C 180,E1 -1994.017,E2 -1994.017} C_VEL
LIN {X 0,Y 580.314,Z 111.008,A -85,B 0,C 180,E1 -1996.914,E2 -1996.914} C_VEL
LIN {X 0,Y 580.29,Z 111.011,A -85,B 0,C 180,E1 -1999.823,E2 -1999.823} C_VEL
LIN {X 0,Y 580.285,Z 111.018,A -85,B 0,C 180,E1 -2001.328,E2 -2001.328} C_VEL
LIN {X 0,Y 579.587,Z 111.099,A -85,B 0,C 180,E1 -2001.907,E2 -2001.907} C_VEL
LIN {X 0,Y 576.708,Z 111.459,A -85,B 0,C 180,E1 -2002.846,E2 -2002.846} C_VEL
LIN {X 0,Y 574.313,Z 111.757,A -85,B 0,C 180,E1 -2003.603,E2 -2003.603} C_VEL
LIN {X 0,Y 573.315,Z 111.878,A -85,B 0,C 180,E1 -2004.187,E2 -2004.187} C_VEL
LIN {X 0,Y 573.25,Z 111.886,A -85,B 0,C 180,E1 -2004.384,E2 -2004.384} C_VEL
LIN {X 0,Y 573.252,Z 111.894,A -85,B 0,C 180,E1 -2006.976,E2 -2006.976} C_VEL
LIN {X 0,Y 573.248,Z 111.888,A -85,B 0,C 180,E1 -2009.488,E2 -2009.488} C_VEL
LIN {X 0,Y 573.254,Z 111.892,A -85,B 0,C 180,E1 -2012.645,E2 -2012.645} C_VEL
LIN {X 0,Y 573.257,Z 111.888,A -85,B 0,C 180,E1 -2015.184,E2 -2015.184} C_VEL
LIN {X 0,Y 573.236,Z 111.888,A -85,B 0,C 180,E1 -2017.808,E2 -2017.808} C_VEL
LIN {X 0,Y 573.246,Z 111.896,A -85,B 0,C 180,E1 -2020.525,E2 -2020.525} C_VEL
LIN {X 0,Y 573.238,Z 111.887,A -85,B 0,C 180,E1 -2023.359,E2 -2023.359} C_VEL
LIN {X 0,Y 573.238,Z 111.892,A -85,B 0,C 180,E1 -2026.641,E2 -2026.641} C_VEL
LIN {X 0,Y 573.246,Z 111.887,A -85,B 0,C 180,E1 -2029.475,E2 -2029.475} C_VEL
LIN {X 0,Y 573.237,Z 111.896,A -85,B 0,C 180,E1 -2032.192,E2 -2032.192} C_VEL
LIN {X 0,Y 573.245,Z 111.887,A -85,B 0,C 180,E1 -2035.228,E2 -2035.228} C_VEL
LIN {X 0,Y 573.242,Z 111.892,A -85,B 0,C 180,E1 -2038.184,E2 -2038.184} C_VEL
LIN {X 0,Y 573.265,Z 111.884,A -85,B 0,C 180,E1 -2040.634,E2 -2040.634} C_VEL
LIN {X 0,Y 573.253,Z 111.886,A -85,B 0,C 180,E1 -2043.024,E2 -2043.024} C_VEL
LIN {X 0,Y 573.276,Z 111.888,A -85,B 0,C 180,E1 -2045.366,E2 -2045.366} C_VEL
LIN {X 0,Y 573.231,Z 111.889,A -85,B 0,C 180,E1 -2048.419,E2 -2048.419} C_VEL
LIN {X 0,Y 573.305,Z 112.069,A -85,B 0,C 180,E1 -2051.145,E2 -2051.145} C_VEL
LIN {X 0,Y 573.31,Z 124.259,A -85,B 0,C 180,E1 -2053.623,E2 -2053.623} C_VEL
LIN {X 0,Y 573.217,Z 138.764,A -85,B 0,C 180,E1 -2056.529,E2 -2056.529} C_VEL
LIN {X 0,Y 573.115,Z 152.051,A -85,B 0,C 180,E1 -2059.134,E2 -2059.134} C_VEL
LIN {X 0,Y 573.312,Z 153.873,A -85,B 0,C 180,E1 -2059.211,E2 -2059.211} C_VEL
LIN {X 0,Y 573.661,Z 160.032,A -85,B 0,C 180,E1 -2059.294,E2 -2059.294} C_VEL
LIN {X 0,Y 573.574,Z 228.415,A -85,B 0,C 180,E1 -2060.167,E2 -2060.167} C_VEL
LIN {X 0,Y 573.527,Z 238.902,A -85,B 0,C 180,E1 -2060.411,E2 -2060.411} C_VEL
LIN {X 0,Y 573.434,Z 250.569,A -85,B 0,C 180,E1 -2060.832,E2 -2060.832} C_VEL
LIN {X 0,Y 573.339,Z 260.964,A -85,B 0,C 180,E1 -2061.364,E2 -2061.364} C_VEL
LIN {X 0,Y 573.257,Z 269.145,A -85,B 0,C 180,E1 -2061.895,E2 -2061.895} C_VEL
LIN {X 0,Y 573.191,Z 276.905,A -85,B 0,C 180,E1 -2062.514,E2 -2062.514} C_VEL
LIN {X 0,Y 573.156,Z 285.137,A -85,B 0,C 180,E1 -2063.323,E2 -2063.323} C_VEL
LIN {X 0,Y 573.113,Z 292.132,A -85,B 0,C 180,E1 -2064.193,E2 -2064.193} C_VEL
LIN {X 0,Y 573.004,Z 297.743,A -85,B 0,C 180,E1 -2065.075,E2 -2065.075} C_VEL
LIN {X 0,Y 573.037,Z 302.955,A -85,B 0,C 180,E1 -2066.132,E2 -2066.132} C_VEL
LIN {X 0,Y 572.992,Z 305.641,A -85,B 0,C 180,E1 -2066.836,E2 -2066.836} C_VEL
LIN {X 0,Y 572.94,Z 308.582,A -85,B 0,C 180,E1 -2067.891,E2 -2067.891} C_VEL
LIN {X 0,Y 572.944,Z 309.872,A -85,B 0,C 180,E1 -2068.594,E2 -2068.594} C_VEL
LIN {X 0,Y 572.936,Z 310.689,A -85,B 0,C 180,E1 -2069.297,E2 -2069.297} C_VEL
LIN {X 0,Y 572.936,Z 310.996,A -85,B 0,C 180,E1 -2070,E2 -2070} C_VEL
LIN {X 0,Y 572.937,Z 310.73,A -85,B 0,C 180,E1 -2070.703,E2 -2070.703} C_VEL
LIN {X 0,Y 572.945,Z 309.996,A -85,B 0,C 180,E1 -2071.406,E2 -2071.406} C_VEL
LIN {X 0,Y 572.94,Z 308.788,A -85,B 0,C 180,E1 -2072.109,E2 -2072.109} C_VEL
LIN {X 0,Y 572.991,Z 305.937,A -85,B 0,C 180,E1 -2073.164,E2 -2073.164} C_VEL
LIN {X 0,Y 573.025,Z 303.345,A -85,B 0,C 180,E1 -2073.868,E2 -2073.868} C_VEL
LIN {X 0,Y 572.983,Z 298.233,A -85,B 0,C 180,E1 -2074.925,E2 -2074.925} C_VEL
LIN {X 0,Y 573.113,Z 292.734,A -85,B 0,C 180,E1 -2075.806,E2 -2075.806} C_VEL
LIN {X 0,Y 573.156,Z 284.345,A -85,B 0,C 180,E1 -2076.849,E2 -2076.849} C_VEL
LIN {X 0,Y 573.217,Z 276.925,A -85,B 0,C 180,E1 -2077.574,E2 -2077.574} C_VEL
LIN {X 0,Y 573.284,Z 269.168,A -85,B 0,C 180,E1 -2078.193,E2 -2078.193} C_VEL
LIN {X 0,Y 573.328,Z 260.99,A -85,B 0,C 180,E1 -2078.725,E2 -2078.725} C_VEL
LIN {X 0,Y 573.434,Z 250.599,A -85,B 0,C 180,E1 -2079.257,E2 -2079.257} C_VEL
LIN {X 0,Y 573.528,Z 238.951,A -85,B 0,C 180,E1 -2079.678,E2 -2079.678} C_VEL
LIN {X 0,Y 573.586,Z 228.489,A -85,B 0,C 180,E1 -2079.922,E2 -2079.922} C_VEL
LIN {X 0,Y 573.64,Z 159.161,A -85,B 0,C 180,E1 -2080.807,E2 -2080.807} C_VEL
LIN {X 0,Y 573.202,Z 152.642,A -85,B 0,C 180,E1 -2080.911,E2 -2080.911} C_VEL
LIN {X 0,Y 573.146,Z 151.459,A -85,B 0,C 180,E1 -2081.047,E2 -2081.047} C_VEL
LIN {X 0,Y 573.227,Z 137.406,A -85,B 0,C 180,E1 -2083.832,E2 -2083.832} C_VEL
LIN {X 0,Y 573.332,Z 123.068,A -85,B 0,C 180,E1 -2086.706,E2 -2086.706} C_VEL
LIN {X 0,Y 573.308,Z 111.968,A -85,B 0,C 180,E1 -2088.974,E2 -2088.974} C_VEL
LIN {X 0,Y 573.229,Z 111.89,A -85,B 0,C 180,E1 -2091.58,E2 -2091.58} C_VEL
LIN {X 0,Y 573.274,Z 111.89,A -85,B 0,C 180,E1 -2094.634,E2 -2094.634} C_VEL
LIN {X 0,Y 573.252,Z 111.887,A -85,B 0,C 180,E1 -2096.976,E2 -2096.976} C_VEL
LIN {X 0,Y 573.246,Z 111.886,A -85,B 0,C 180,E1 -2099.488,E2 -2099.488} C_VEL
LIN {X 0,Y 573.253,Z 111.888,A -85,B 0,C 180,E1 -2102.645,E2 -2102.645} C_VEL
LIN {X 0,Y 573.254,Z 111.885,A -85,B 0,C 180,E1 -2105.184,E2 -2105.184} C_VEL
LIN {X 0,Y 573.236,Z 111.894,A -85,B 0,C 180,E1 -2107.807,E2 -2107.807} C_VEL
LIN {X 0,Y 573.244,Z 111.888,A -85,B 0,C 180,E1 -2110.525,E2 -2110.525} C_VEL
LIN {X 0,Y 573.236,Z 111.891,A -85,B 0,C 180,E1 -2113.359,E2 -2113.359} C_VEL
LIN {X 0,Y 573.244,Z 111.887,A -85,B 0,C 180,E1 -2116.331,E2 -2116.331} C_VEL
LIN {X 0,Y 573.238,Z 111.887,A -85,B 0,C 180,E1 -2118.544,E2 -2118.544} C_VEL
LIN {X 0,Y 573.241,Z 111.894,A -85,B 0,C 180,E1 -2121.298,E2 -2121.298} C_VEL
LIN {X 0,Y 573.245,Z 111.887,A -85,B 0,C 180,E1 -2124.014,E2 -2124.014} C_VEL
LIN {X 0,Y 573.268,Z 111.884,A -85,B 0,C 180,E1 -2126.518,E2 -2126.518} C_VEL
LIN {X 0,Y 573.229,Z 111.897,A -85,B 0,C 180,E1 -2129.117,E2 -2129.117} C_VEL
LIN {X 0,Y 573.251,Z 111.886,A -85,B 0,C 180,E1 -2131.971,E2 -2131.971} C_VEL
LIN {X 0,Y 573.252,Z 111.89,A -85,B 0,C 180,E1 -2134.59,E2 -2134.59} C_VEL
LIN {X 0,Y 573.236,Z 111.888,A -85,B 0,C 180,E1 -2137.662,E2 -2137.662} C_VEL
LIN {X 0,Y 573.277,Z 111.892,A -85,B 0,C 180,E1 -2140.728,E2 -2140.728} C_VEL
LIN {X 0,Y 573.251,Z 111.886,A -85,B 0,C 180,E1 -2143.622,E2 -2143.622} C_VEL
LIN {X 0,Y 573.272,Z 111.884,A -85,B 0,C 180,E1 -2145.807,E2 -2145.807} C_VEL
LIN {X 0,Y 573.262,Z 111.889,A -85,B 0,C 180,E1 -2148.745,E2 -2148.745} C_VEL
LIN {X 0,Y 573.284,Z 111.882,A -85,B 0,C 180,E1 -2151.54,E2 -2151.54} C_VEL
LIN {X 0,Y 573.29,Z 111.887,A -85,B 0,C 180,E1 -2154.372,E2 -2154.372} C_VEL
LIN {X 0,Y 573.314,Z 111.885,A -85,B 0,C 180,E1 -2157.892,E2 -2157.892} C_VEL
LIN {X 0,Y 573.33,Z 111.876,A -85,B 0,C 180,E1 -2160.702,E2 -2160.702} C_VEL
LIN {X 0,Y 573.303,Z 111.879,A -85,B 0,C 180,E1 -2162.811,E2 -2162.811} C_VEL
LIN {X 0,Y 573.289,Z 111.888,A -85,B 0,C 180,E1 -2165.628,E2 -2165.628} C_VEL
LIN {X 0,Y 573.284,Z 111.882,A -85,B 0,C 180,E1 -2168.459,E2 -2168.459} C_VEL
LIN {X 0,Y 573.27,Z 111.889,A -85,B 0,C 180,E1 -2171.312,E2 -2171.312} C_VEL
LIN {X 0,Y 573.272,Z 111.883,A -85,B 0,C 180,E1 -2174.193,E2 -2174.193} C_VEL
LIN {X 0,Y 573.257,Z 111.891,A -85,B 0,C 180,E1 -2177.112,E2 -2177.112} C_VEL
LIN {X 0,Y 573.251,Z 111.886,A -85,B 0,C 180,E1 -2180.077,E2 -2180.077} C_VEL
LIN {X 0,Y 573.233,Z 111.898,A -85,B 0,C 180,E1 -2183.099,E2 -2183.099} C_VEL
LIN {X 0,Y 573.251,Z 111.889,A -85,B 0,C 180,E1 -2185.41,E2 -2185.41} C_VEL
LIN {X 0,Y 573.25,Z 111.886,A -85,B 0,C 180,E1 -2188.029,E2 -2188.029} C_VEL
LIN {X 0,Y 573.245,Z 111.888,A -85,B 0,C 180,E1 -2190.176,E2 -2190.176} C_VEL
LIN {X 0,Y 573.252,Z 111.894,A -85,B 0,C 180,E1 -2192.645,E2 -2192.645} C_VEL
LIN {X 0,Y 573.253,Z 111.887,A -85,B 0,C 180,E1 -2195.185,E2 -2195.185} C_VEL
LIN {X 0,Y 573.234,Z 111.888,A -85,B 0,C 180,E1 -2197.808,E2 -2197.808} C_VEL
LIN {X 0,Y 573.243,Z 111.895,A -85,B 0,C 180,E1 -2200.525,E2 -2200.525} C_VEL
LIN {X 0,Y 573.238,Z 111.887,A -85,B 0,C 180,E1 -2203.359,E2 -2203.359} C_VEL
LIN {X 0,Y 573.237,Z 111.895,A -85,B 0,C 180,E1 -2206.332,E2 -2206.332} C_VEL
LIN {X 0,Y 573.232,Z 111.891,A -85,B 0,C 180,E1 -2208.543,E2 -2208.543} C_VEL
LIN {X 0,Y 573.24,Z 111.888,A -85,B 0,C 180,E1 -2211.299,E2 -2211.299} C_VEL
LIN {X 0,Y 573.238,Z 111.895,A -85,B 0,C 180,E1 -2214.015,E2 -2214.015} C_VEL
LIN {X 0,Y 573.238,Z 111.888,A -85,B 0,C 180,E1 -2216.516,E2 -2216.516} C_VEL
LIN {X 0,Y 573.227,Z 111.89,A -85,B 0,C 180,E1 -2219.118,E2 -2219.118} C_VEL
LIN {X 0,Y 573.252,Z 111.889,A -85,B 0,C 180,E1 -2221.971,E2 -2221.971} C_VEL
LIN {X 0,Y 573.246,Z 111.886,A -85,B 0,C 180,E1 -2224.59,E2 -2224.59} C_VEL
LIN {X 0,Y 573.233,Z 111.892,A -85,B 0,C 180,E1 -2227.662,E2 -2227.662} C_VEL
LIN {X 0,Y 573.314,Z 112.044,A -85,B 0,C 180,E1 -2228.822,E2 -2228.822} C_VEL
LIN {X 0,Y 573.581,Z 117.127,A -85,B 0,C 180,E1 -2229.749,E2 -2229.749} C_VEL
LIN {X 0,Y 573.46,Z 134.021,A -85,B 0,C 180,E1 -2232.711,E2 -2232.711} C_VEL
LIN {X 0,Y 573.314,Z 150.464,A -85,B 0,C 180,E1 -2235.564,E2 -2235.564} C_VEL
LIN {X 0,Y 573.192,Z 167.571,A -85,B 0,C 180,E1 -2238.507,E2 -2238.507} C_VEL
LIN {X 0,Y 573.188,Z 171.337,A -85,B 0,C 180,E1 -2239.106,E2 -2239.106} C_VEL
LIN {X 0,Y 573.621,Z 175.3,A -85,B 0,C 180,E1 -2239.189,E2 -2239.189} C_VEL
LIN {X 0,Y 573.582,Z 247.151,A -85,B 0,C 180,E1 -2240.101,E2 -2240.101} C_VEL
LIN {X 0,Y 573.511,Z 256.419,A -85,B 0,C 180,E1 -2240.3,E2 -2240.3} C_VEL
LIN {X 0,Y 573.457,Z 264.892,A -85,B 0,C 180,E1 -2240.566,E2 -2240.566} C_VEL
LIN {X 0,Y 573.412,Z 273.398,A -85,B 0,C 180,E1 -2240.921,E2 -2240.921} C_VEL
LIN {X 0,Y 573.341,Z 281.73,A -85,B 0,C 180,E1 -2241.364,E2 -2241.364} C_VEL
